# B&R Automation Studio project RS15_RX_30005_r00 (part 4)

#### A2_CycleCyclic.st
```iecst
(********************************************************************
 * COPYRIGHT -- .
 ********************************************************************
 * Program: A2_Cycle
 * File: A2_CycleCyclic.st
 * Author: Dominique
 * Created: October 15, 2011
 ********************************************************************
 * Implementation of program A2_Cycle
 ********************************************************************)

PROGRAM _CYCLIC

// Manu axis movement for timing setting

    //----------------------------------------------------------------------
    // FP Nip rolle auto Off
    // During timing setting automatique switch Off nip rolle
       stTON_02 (IN:=gstCycA[2].CycManTimSet.bCyc ,PT:=T#650ms) ;
       stTOF_00 (IN:=gstCycA[2].CycManTimSet.bCyc ,PT:=T#1s_500ms) ;
       g_bFP_NipRolAutoOff := gstCycA[2].CycManTimSet.bCyc OR
                              stTOF_00.Q                   ;

    //----------------------------------------------------------------------
    // Offset management

    // When synchro is off, Offset is set to 0
       IF NOT(gA[2].Ind_SynchronizedMotion) AND
          gstCycA[2].CycManTimSet.bFCyc     THEN
         rPrintRolActOffsetInch := 0.0 ;
         rSP_PrintRolOffsetInch := 0.0 ;
       END_IF ;
    // Set point Offset value Lock
    g_bLockSP_OffsetPrintRol := NOT(g_bCondManuTimSet)            OR
                                gstCycA[2].CycManTimSet.bSCyc     OR
                                0                                 ;

    // Offset Manu button animation
    bLockOffsetPB_Man := g_bFP_SP_Offset                   OR
                         g_bStartOffsetAuto                OR
                         NOT(g_bCondManuTimSet)            ;

    // Limit offset set point
    rSP_PrintRolOffsetInch := LIMIT(0.0,rSP_PrintRolOffsetInch,gRecipeActive.Repeat) ;
    IF gA[2].Cmd_ManuTimSetPlus THEN
      rSP_PrintRolOffsetInch := 0.0 ;
    END_IF ;
    // Calculation distance on axis
    rSP_AxisOffsetInch := rSP_PrintRolOffsetInch * gA[2].rRSynNum / gA[2].rRSynDen ;

    // Offset Auto button animation
    bLockOffsetPB := gstCycA[2].CycManTimSet.bFCyc     AND
                     (rSP_PrintRolOffsetInch <= 0.0)   OR
                     g_HMI_Cmd_ManuTimSetPlus          OR
                     (gstCycA[2].CycManTimSet.iStep>2) AND
                     NOT(g_bFP_SP_Offset)            ;

    IF NOT(bLockOffsetPB)        AND
       NOT(HMI_Cmd_AutoOffsetPB) THEN
      iAnimOffsetPB := 2 ;                     // Ready
    END_IF ;
    IF (rSP_PrintRolOffsetInch>0.0) AND
       NOT(g_bFP_SP_Offset)         AND
       NOT(bLockOffsetPB)           AND
       HMI_Cmd_AutoOffsetPB         THEN
      iAnimOffsetPB := 3 ;                     // Start
    END_IF ;
    IF g_bFP_SP_Offset THEN
      iAnimOffsetPB := 4 ;                     // Stop
    END_IF ;
    IF bLockOffsetPB THEN
      iAnimOffsetPB := 0 ;                     // PB Lock
    END_IF ;

    CASE iAnimOffsetPB OF
      0..1 : ; // PB Lock
        uiSP_OffsetCol_Ind := gBlue + gWhite * 256 ;
      2 : ;    // Ready
        uiSP_OffsetCol_Ind := gBlue + gWhite * 256 ;
      3 : ;    // Start
        uiSP_OffsetCol_Ind := gGreen + gBlack * 256 ;
      4 : ;    // Stop
        uiSP_OffsetCol_Ind := gRed + gBlack * 256 ;
    END_CASE
    uiSP_OffsetTxt_Ind := iAnimOffsetPB ;

    // Start Offset Auto
    IF EDGENEG(HMI_Cmd_AutoOffsetPB) THEN
      g_bStartOffsetAuto := 1 ;
    END_IF ;

    //---------------------------------------------------------------------------------------------------------------------
    // Printing rolle offset cycle
    //---------------------------------------------------------------------------------------------------------------------
    // Start cycle
    gstCycA[2].CycManTimSet.CmdStart := ( gA[2].Cmd_ManuTimSetPlus    OR
                                          gA[2].Cmd_ManuTimSetMinus ) AND
                                        gA[2].Ind_Ready               OR
                                        g_bStartOffsetAuto            AND
                                        1                             ;
    IF gstCycA[2].CycManTimSet.CmdStart THEN
      gstCycA[2].CycManTimSet.bSCyc := 1 ;
    END_IF ;

    //----------------------------------------------------------------------
    // Cycle at rest
    IF NOT(gstCycA[2].CycManTimSet.bSCyc) AND
       1                                  THEN
      IF NOT( gstCycA[2].CycManTimSet.bFCyc ) THEN
        // Init after cycle unpropaly ended
        gstCycA[2].CycManTimSet.bFCyc := 1 ;
        gstCycA[2].CycManTimSet.bCyc  := 0 ;

        g_bFP_SP_Offset                      := 0 ;
        g_bStartOffsetAuto                   := 0 ;
        gstCycA[2].CycManTimSet.CmdMov       := 0 ;
        gstCycA[2].CycManTimSet.CmdStop      := 0 ;
        gstCycA[2].CycManTimSet.CmdSynchroOn := 0 ;
        gstCycA[2].CycManTimSet.CmdExeMov    := 0 ;
        gstCycA[2].CycManTimSet.CmdExeStop   := 0 ;
      END_IF
      gstCycA[2].CycManTimSet.iStep := 0 ;
      RETURN ;
    ELSE
    //----------------------------------------------------------------------
    // Cycle running

      // Permanent conditions
      IF ( NOT(gA[2].Ind_Ready)                    OR
           NOT(gstCycA[2].CycManTimSet.CmdStart) ) AND
         NOT(g_bFP_SP_Offset)                      AND
         NOT(g_bStartOffsetAuto)                   AND
         (gstCycA[2].CycManTimSet.iStep <= 2)      THEN
        gstCycA[2].CycManTimSet.bSCyc := 0 ;
        RETURN ;
      END_IF

      IF g_bFP_SP_Offset                   AND
         ( NOT(gStopStringOK)              OR
           EDGEPOS(HMI_Cmd_AutoOffsetPB) ) THEN
        gstCycA[2].CycManTimSet.iStep := C_iSTEP_13 ;
        // Action Step 13
        gstCycA[2].CycManTimSet.CmdExeMov  := 0 ;
        gstCycA[2].CycManTimSet.CmdExeStop := 1 ;
        // Waiting Stop
      END_IF

      IF (gstCycA[2].CycManTimSet.iStep = C_iSTEP_11) AND
         (gstCycA[2].CycManTimSet.enMoveStat = FAULT) THEN
        gstCycA[2].CycManTimSet.iStep := C_iSTEP_16 ;
        // Action Step 16
        // Waiting Reset Fault
      END_IF

      // Permanent actions
      stTON_01 (
            IN := ( gstCycA[2].CycManTimSet.iStep = C_iSTEP_0 ) ,
            PT := T#30ms
               ) ;

      // Actual offset calculation
      IF (gstCycA[2].CycManTimSet.iStep >= C_iSTEP_3) THEN
        rTempDiffPrintRolPos := g_rPrintRolCalcPos_in - rMemoPosPrintRol ;
        rMemoPosPrintRol := g_rPrintRolCalcPos_in ;
        rDiffPrintRolPos := H_FC_Modulus (
                                 IN_rMod := gRecipeActive.Repeat ,
                                 IN_rVar := rTempDiffPrintRolPos
                                         ) ;
        rTempActOffsetInch[2] := rPrintRolActOffsetInch ;
        rPrintRolActOffsetInch := rPrintRolActOffsetInch + rDiffPrintRolPos ;
        rPrintRolActOffsetInch := H_FC_Modulus (
                                       IN_rMod := gRecipeActive.Repeat ,
                                       IN_rVar := rPrintRolActOffsetInch
                                               ) ;

        // Set point distance Offset animation
        IF g_bFP_SP_Offset THEN
          rSP_PrintRolOffsetInch := rSP_PrintRolOffsetInch - rDiffPrintRolPos ;
          IF (rSP_PrintRolOffsetInch < 0.001) THEN
            rSP_PrintRolOffsetInch := 0.0 ;
          END_IF
        END_IF
      END_IF

      stTON_03 (
            IN := (gstCycA[2].CycManTimSet.iStep = C_iSTEP_15) AND NOT(HMI_Cmd_AutoOffsetPB) ,
            PT := T#500ms
               ) ;

    END_IF
    //----------------------------------------------------------------------
    // Cycle steps

        CASE gstCycA[2].CycManTimSet.iStep OF

        C_iSTEP_0 :
         //----------------------------------------------
         // Etape 1 : Initialisation
         //           Waiting auto switch Off nip rolle
         //----------------------------------------------
          IF stTON_01.Q THEN
            gstCycA[2].CycManTimSet.iStep := C_iSTEP_1 ;

            // Action Step 1
            gstCycA[2].CycManTimSet.bFCyc := 0 ;
            gstCycA[2].CycManTimSet.bCyc  := 1 ;

            gstCycA[2].CycManTimSet.rSP_Distance := 0 ;
          END_IF

        C_iSTEP_1 :
         //----------------------------------------------
         // Etape 2  : Synchro
         //----------------------------------------------
          // Condition Step2
          IF (stTON_02.Q OR stTOF_00.Q) THEN
            gstCycA[2].CycManTimSet.iStep := C_iSTEP_2 ;

            // Action Step 2
            gstCycA[2].CycManTimSet.CmdSynchroOn := 1 ;
          END_IF

        C_iSTEP_2 :
         //----------------------------------------------
         // Step 3 : Activation motion and Stop waiting
         // Etape 10 : Synchro and start Offset with set point
         //----------------------------------------------
          IF gstCycA[2].CycManTimSet.bSynchroOkSlavA[2] AND
             (rSP_PrintRolOffsetInch <= 0)              THEN
            gstCycA[2].CycManTimSet.iStep := C_iSTEP_3 ;

            // Action Step 3
            gstCycA[2].CycManTimSet.CmdMov  := 1 ;
            gstCycA[2].CycManTimSet.CmdStop := 0 ;
            // Stop waiting
            // Memo printing cylinder actual position
            rMemoPosPrintRol := g_rPrintRolCalcPos_in ;
            RETURN ;
          END_IF
          // Condition Step10
          IF stTON_02.Q                                 AND
             gstCycA[2].CycManTimSet.bSynchroOkSlavA[2] AND
             g_bStartOffsetAuto                         AND
             ( gstCycA[2].CycManTimSet.bTestOn          OR
               NOT(gstCycA[2].CycManTimSet.bModTest) )  THEN
            gstCycA[2].CycManTimSet.iStep := C_iSTEP_10 ;

            // Action Step 10
            gstCycA[2].CycManTimSet.bTestOn := 0 ;

            g_bFP_SP_Offset    := 1 ;
            g_bStartOffsetAuto := 0 ;
            gstCycA[2].CycManTimSet.CmdExeMov  := 1 ;
            gstCycA[2].CycManTimSet.CmdExeStop := 0 ;
            gstCycA[2].CycManTimSet.rSP_Distance := rSP_AxisOffsetInch ;
            // Memo printing cylinder actual position
            rMemoPosPrintRol := g_rPrintRolCalcPos_in ;
          END_IF

        C_iSTEP_3 :
         //----------------------------------------------
         // Step 4 : Stop motion and End stop waiting
         //----------------------------------------------
          IF NOT(gstCycA[2].CycManTimSet.CmdStart) THEN
            gstCycA[2].CycManTimSet.iStep := C_iSTEP_4 ;

            // Action Step 4
            gstCycA[2].CycManTimSet.CmdMov  := 0 ;
            gstCycA[2].CycManTimSet.CmdStop := 1 ;
            // End stop waiting
          END_IF

        C_iSTEP_4 :
         //----------------------------------------------
         // Step 3 : Activation motion and Stop waiting
         // Step 5 : Cut synchro
         //----------------------------------------------
          // Condition Step3
          IF gstCycA[2].CycManTimSet.CmdStart THEN
            gstCycA[2].CycManTimSet.iStep := C_iSTEP_3 ;

            // Action Step 3
            gstCycA[2].CycManTimSet.CmdMov  := 1 ;
            gstCycA[2].CycManTimSet.CmdStop := 0 ;
            // Stop waiting
            RETURN ;
          END_IF ;
          // Condition Step5
          IF NOT(gstCycA[2].CycManTimSet.CmdStop) THEN
            gstCycA[2].CycManTimSet.iStep := C_iSTEP_5 ;

            // Action Step 5
            gstCycA[2].CycManTimSet.CmdSynchroOn := 0 ;
          END_IF

        C_iSTEP_5 :
         //----------------------------------------------
         // Step 0 : First step
         //----------------------------------------------
          IF TRUE THEN
            gstCycA[2].CycManTimSet.iStep := C_iSTEP_0 ;

            // Action Step 0
            gstCycA[2].CycManTimSet.bSCyc := 0 ;
            gstCycA[2].CycManTimSet.bFCyc := 1 ;
            gstCycA[2].CycManTimSet.bCyc  := 0 ;
          END_IF

        C_iSTEP_10 :
         //----------------------------------------------
         // Step 11 : Waiting end of move
         //----------------------------------------------
          IF TRUE                                          AND
             ( gstCycA[2].CycManTimSet.bTestOn             OR
               NOT(gstCycA[2].CycManTimSet.bModTest) )     THEN
            gstCycA[2].CycManTimSet.iStep := C_iSTEP_11 ;

            // Action Step 11
            gstCycA[2].CycManTimSet.bTestOn := 0 ;

            // Waiting end of move
          END_IF

        C_iSTEP_11 :
         //----------------------------------------------
         // Step 12 : End move
         //----------------------------------------------
          IF (gstCycA[2].CycManTimSet.enMoveStat = FINISHED) AND
             ( gstCycA[2].CycManTimSet.bTestOn               OR
               NOT(gstCycA[2].CycManTimSet.bModTest) )       THEN
            gstCycA[2].CycManTimSet.iStep := C_iSTEP_12 ;

            // Action Step 12
            gstCycA[2].CycManTimSet.bTestOn := 0 ;

            gstCycA[2].CycManTimSet.CmdExeMov := 0 ;
            g_bFP_SP_Offset := 0 ;
          END_IF

        C_iSTEP_12 :
         //----------------------------------------------
         // Step 0 : First step
         //----------------------------------------------
          IF (gstCycA[2].CycManTimSet.enMoveStat = INACTIVE) AND
             ( gstCycA[2].CycManTimSet.bTestOn               OR
               NOT(gstCycA[2].CycManTimSet.bModTest) )       THEN
            gstCycA[2].CycManTimSet.iStep := C_iSTEP_0 ;

            // Action Step 0
            gstCycA[2].CycManTimSet.bTestOn := 0 ;

            gstCycA[2].CycManTimSet.CmdSynchroOn := 0 ;

            gstCycA[2].CycManTimSet.bSCyc := 0 ;
            gstCycA[2].CycManTimSet.bFCyc := 1 ;
            gstCycA[2].CycManTimSet.bCyc  := 0 ;
          END_IF

        C_iSTEP_13 :
         //----------------------------------------------
         // Step 14 : End stop
         //----------------------------------------------
          IF (gstCycA[2].CycManTimSet.enMoveStat = INACTIVE) AND
             ( gstCycA[2].CycManTimSet.bTestOn               OR
               NOT(gstCycA[2].CycManTimSet.bModTest) )       AND
             gA[2].Ind_StandStill                            THEN
            gstCycA[2].CycManTimSet.iStep := C_iSTEP_14 ;

            // Action Step 14
            gstCycA[2].CycManTimSet.bTestOn := 0 ;

            gstCycA[2].CycManTimSet.CmdExeStop := 0 ;
          END_IF

        C_iSTEP_14 :
         //----------------------------------------------
         // Step 15 : Waiting
         //----------------------------------------------
          IF gA[2].Ind_SynchronizedMotion                  AND
             ( gstCycA[2].CycManTimSet.bTestOn             OR
               NOT(gstCycA[2].CycManTimSet.bModTest) )     THEN
            gstCycA[2].CycManTimSet.iStep := C_iSTEP_15 ;

            // Action Step 15
            gstCycA[2].CycManTimSet.bTestOn := 0 ;

            // Waiting
          END_IF

        C_iSTEP_15 :
         //----------------------------------------------
         // Step 0 : First step
         //----------------------------------------------
          IF stTON_03.Q                                    AND
             ( gstCycA[2].CycManTimSet.bTestOn             OR
               NOT(gstCycA[2].CycManTimSet.bModTest) )     THEN
            gstCycA[2].CycManTimSet.iStep := C_iSTEP_0 ;

            // Action Step 0
            gstCycA[2].CycManTimSet.bTestOn := 0 ;

            gstCycA[2].CycManTimSet.bSCyc := 0 ;
            gstCycA[2].CycManTimSet.bFCyc := 1 ;
            gstCycA[2].CycManTimSet.bCyc  := 0 ;
            g_bStartOffsetAuto := 0 ;
            g_bFP_SP_Offset    := 0 ;
            gstCycA[2].CycManTimSet.CmdSynchroOn := 0 ;
          END_IF

        C_iSTEP_16 :
         //----------------------------------------------
         // Step 17 : End cycle
         //----------------------------------------------
          IF gAlarmReset                                   AND
             ( gstCycA[2].CycManTimSet.bTestOn             OR
               NOT(gstCycA[2].CycManTimSet.bModTest) )     THEN
            gstCycA[2].CycManTimSet.iStep := C_iSTEP_17 ;

            // Action Step 17
            gstCycA[2].CycManTimSet.bTestOn := 0 ;

            gstCycA[2].CycManTimSet.CmdExeMov := 0 ;
          END_IF

        C_iSTEP_17 :
         //----------------------------------------------
         // Step 0 : First step
         //----------------------------------------------
          IF (gstCycA[2].CycManTimSet.enMoveStat = INACTIVE) AND
             ( gstCycA[2].CycManTimSet.bTestOn               OR
               NOT(gstCycA[2].CycManTimSet.bModTest) )       THEN
            gstCycA[2].CycManTimSet.iStep := C_iSTEP_0 ;

            // Action Step 0
            gstCycA[2].CycManTimSet.bTestOn := 0 ;

            gstCycA[2].CycManTimSet.bSCyc := 0 ;
            gstCycA[2].CycManTimSet.bFCyc := 1 ;
            gstCycA[2].CycManTimSet.bCyc  := 0 ;
            g_bStartOffsetAuto := 0 ;
            g_bFP_SP_Offset    := 0 ;
            gstCycA[2].CycManTimSet.CmdSynchroOn := 0 ;
          END_IF
        END_CASE
    //---------------------------------------------------------------------------------------------------------------------

END_PROGRAM
```

### Package Logical/BagMachine_Section/Holding - Axis

### Data object Logical/BagMachine_Section/Holding/Axis3/A3_Init (Ax) - Servo Axis Initialization File

#### A3_Init.ax
```
InitParameter (Version=2.24.0, NcSwId=ACP10)
  ACP10AXIS_typ:
    dig_in:
      level:
        reference = ncACTIV_HI
        pos_hw_end = ncACTIV_HI
        neg_hw_end = ncACTIV_HI
        trigger1 = ncACTIV_HI
        trigger2 = ncACTIV_HI
    encoder_if:
      parameter:
        count_dir = ncINVERSE
        scaling:
          load:
            units = 24000  // Units at the load = 36000 x 2 / 3
            rev_motor = 1  // Motor revolutions = 1
    limit:
      parameter:
        v_pos = 1.2e+006
        v_neg = 1.2e+006
        a1_pos = 5e+006
        a2_pos = 5e+006
        a1_neg = 5e+006
        a2_neg = 5e+006
        t_jolt = 0.0
        t_in_pos = 0.0
        pos_sw_end = 8388607
        neg_sw_end = -8388608
        ds_warning = 500.0
        ds_stop = 1000.0
        a_stop = 1e+030
        dv_stop = 0
        dv_stop_mode = ncOFF
    controller:
      mode = ncPOSITION
      position:
        kv = 300.0
        tn = 0.0
        t_predict = 0.0004
        t_total = 0.0012
        p_max = 1e+030
        i_max = 0.0
      speed:
        kv = 30.0
        tn = 0.0
        t_filter = 0.0
        isq_filter1:
          type = ncOFF
          a0 = 0.0
          a1 = 0.0
          b0 = 0.0
          b1 = 0.0
          b2 = 0.0
          c0_par_id = 0
          c1_par_id = 0
        isq_filter2:
          type = ncOFF
          a0 = 0.0
          a1 = 0.0
          b0 = 0.0
          b1 = 0.0
          b2 = 0.0
          c0_par_id = 0
          c1_par_id = 0
        isq_filter3:
          type = ncOFF
          a0 = 0.0
          a1 = 0.0
          b0 = 0.0
          b1 = 0.0
          b2 = 0.0
          c0_par_id = 0
          c1_par_id = 0
      uf:
        type = ncLINEAR
        auto_config = ncMOTOR_PAR
        u0 = 0.0
        un = 0.0
        fn = 50.0
        k_f_slip = 0.0
      ff:
        torque_load = 0.0
        torque_pos = 0.0
        torque_neg = 0.0
        kv_torque = 0.0
        inertia = 0.0
        t_filter_a = 0.0
    move:
      stop:
        parameter[0]:
          decel_ramp = ncA_LIMIT
          controller = ncON
        parameter[1]:
          decel_ramp = ncA_LIMIT
          controller = ncON
        parameter[2]:
          decel_ramp = ncA_LIMIT
          controller = ncON
        parameter[3]:
          decel_ramp = ncA_LIMIT
          controller = ncON
        quickstop:
          decel_ramp = ncA_LIMIT
        drive_error:
          decel_ramp = ncA_LIMIT
      homing:
        parameter:
          s = 0
          v_switch = 3600.0
          v_trigger = 360.0
          a = 50000.0
          mode = ncHOME_OFFSET
          edge_sw = ncNEGATIVE
          start_dir = ncNEGATIVE
          trigg_dir = ncNEGATIVE
          ref_pulse = ncOFF
          tr_s_block = 0.0
      basis:
        parameter:
          v_pos = 36000.0
          v_neg = 100000.0
          a1_pos = 50000.0
          a2_pos = 50000.0
          a1_neg = 50000.0
          a2_neg = 50000.0
    message:
      text:
        parameter:
          format = ncBREAK
          columns = 80
          data_modul = Error_Eng
```

### Data object Logical/BagMachine_Section/Holding/Axis3/A3_Par (Apt) - Servo Axis Parameter File

#### A3_Par.apt
```
AcoposParameterTable:
  Root Parameters:
    110 = ncSW_OFF (Name=CMD_SIMULATION)  // Simulation mode: Command
    128 = 1 (Name=SGEN_SW_END_IGNORE)  // SGEN_SW_END_IGNORE
    390 = 565 (Name=UDC_NOMINAL, Unit=V)  // CTRL DC bus: Nominal voltage
    944 = 464 (Name=REFERENCE_SWITCH_PARID)  // REFERENCE_SWITCH_PARID
```

### Program Logical/BagMachine_Section/Holding/Axis3/A3_Basic (IEC) - Basic Servo

#### A3_Basic.var - Local variables
```iecst
(********************************************************************
 * COPYRIGHT -- Microsoft
 ********************************************************************
 * Program: A3_Basic
 * File: A3_Basic.var
 * Author: pkiel
 * Created: July 13, 2011
 ********************************************************************
 * Local variables of program A3_Basic
 ********************************************************************)
VAR
	AutoAck : BOOL;
	AxisErrorNcAccess : UINT;
	DriveStatus : MC_DRIVESTATUS_TYP;
	HomeRestore : BOOL;
	InitEndlessPosition : BOOL;
	InitModPos_Done : BOOL;
	InitModPosition : BOOL;
	MC_BR_InitEndlessPosition_0 : MC_BR_InitEndlessPosition;
	MC_BR_InitModPos_0 : MC_BR_InitModPos;
  MC_BR_Phasing_0 : MC_BR_Phasing;
  MC_BR_Phasing_1 : MC_BR_Phasing;
	MC_BR_ReadDriveStatus_0 : MC_BR_ReadDriveStatus;
	MC_Home_0 : MC_Home;
	MC_Home_1 : MC_Home;
	MC_MoveVelocity_0 : MC_MoveVelocity;
	MC_Power_0 : MC_Power;
	MC_ReadActualPosition_0 : MC_ReadActualPosition;
	MC_ReadActualTorque_0 : MC_ReadActualTorque;
	MC_ReadActualVelocity_0 : MC_ReadActualVelocity;
	MC_ReadAxisError_0 : MC_ReadAxisError;
	MC_ReadStatus_0 : MC_ReadStatus;
	MC_Reset_0 : MC_Reset;
  MC_Stop_0 : MC_Stop;
  MC_Stop_1 : MC_Stop;

  MC_SetOverride_0 : MC_SetOverride ;
	ResetError : BOOL;
  rAxisTimSet_SP_Vel  : REAL ; (*Set point Velocity for Axis manual timing setting cycle, in units/s*)
  rAxisTimSet_SP_Acc  : REAL ; (*Set point Acceleration for Axis manual timing setting cycle, in units/s²*)
  rAxisTimSet_SP_Dec  : REAL ; (*Set point Deceleration for Axis manual timing setting cycle, in units/s²*)
  uiAxisTimSet_SP_Dir : USINT ; (*Set point Direction for Axis manual timing setting cycle*)
  uiAxisTimSet_SP_ShiftAppMode : UINT ; (*Set point Shit Application mode for phasing Axis manual timing setting cycle*)
  bTest_ : ARRAY[0..9] OF  BOOL;
  iTest_ : ARRAY[0..9] OF  INT;
  rTemp_ : ARRAY[0..9] OF REAL ;
  rTempActPhasDeg : REAL ;
  rTempActPhasDeg1 : REAL ;
  rTempActPhasDeg2 : REAL ;
  rTempAxisTimSet_SP_Acc : REAL;
  rTempAxisTimSet_SP_Dec : REAL;
  rPhasing_1_SP_Acc : REAL;
  rA9PosCorDeg  : REAL;
  rRepeatMetric : REAL;

  iiSP_SlPos_U  : DINT ; (*On Slave side, input set point position of the position controller ParID 428, in unit*)
  rSP_SlPos_Deg : REAL ; (*On Slave side, input set point position of the position controller ParID 428, in deg*)
  iiSP_MaPos_U  : DINT ; (*On Master side, input set point position of the position controller ParID 412, in unit*)
  rSP_MaPos_Deg : REAL ; (*On Master side, input set point position of the position controller ParID 412, in deg*)
  MC_BR_CyclicRead_0 : MC_BR_CyclicRead ;
  MC_BR_CyclicRead_1 : MC_BR_CyclicRead ;

  H_FB_RelativeChangeLimitReal_0 : H_FB_RelativeChangeLimitReal;
  rMin : REAL;
  IN_rRepeat : REAL;
  IN_rMin : REAL;
  IN_rMax : REAL;
  IN_bEnable : BOOL;
  rDiff : REAL;
  INOUT_rLimitIn : REAL;
  rOldLimitIn : REAL;
  rMax : REAL;
  rInput : REAL;
  IN_rInput : REAL;
  rOld : REAL;
  OUT_bChange : BOOL;
  OUT_rDiff : REAL;
  OUT_bOK : BOOL ;
  iIndex : INT ;
  rTempPosHolding : REAL ;
  st_TON_0 : TON;
  rSP_ShiftHolding   : REAL ;
  rSP_PhaseOffset    : REAL ;
  rSP_PhaseOffsetVal : REAL ;

  rA3PosTempAxis_deg : REAL ;
END_VAR
```

### Program Logical/BagMachine_Section/Holding/Axis3/A3_Control (IEC) - Servo Control

#### A3_Control.var
```iecst
(********************************************************************
 * COPYRIGHT -- Microsoft
 ********************************************************************
 * Program: A3_Control
 * File: A3_Control.var
 * Author: pkiel
 * Created: July 13, 2011
 ********************************************************************
 * Local variables of program A3_Control
 ********************************************************************)
VAR
	HGW_ChangeReal_0 : HGW_ChangeReal;
	HGW_RelativeChangeReal_0 : HGW_RelativeChangeReal;
  H_FB_RelativeChangeLimitReal1_0 : H_FB_RelativeChangeLimitReal1;
	HGW_Toggle_0 : HGW_Toggle;
	Synch_Permissive : BOOL;
	TOF_0 : TOF;
	TON_0 : TON;
  rIncrOffsetAxeRun_Inch : REAL ;
END_VAR
```

#### A3_ControlCyclic.ld
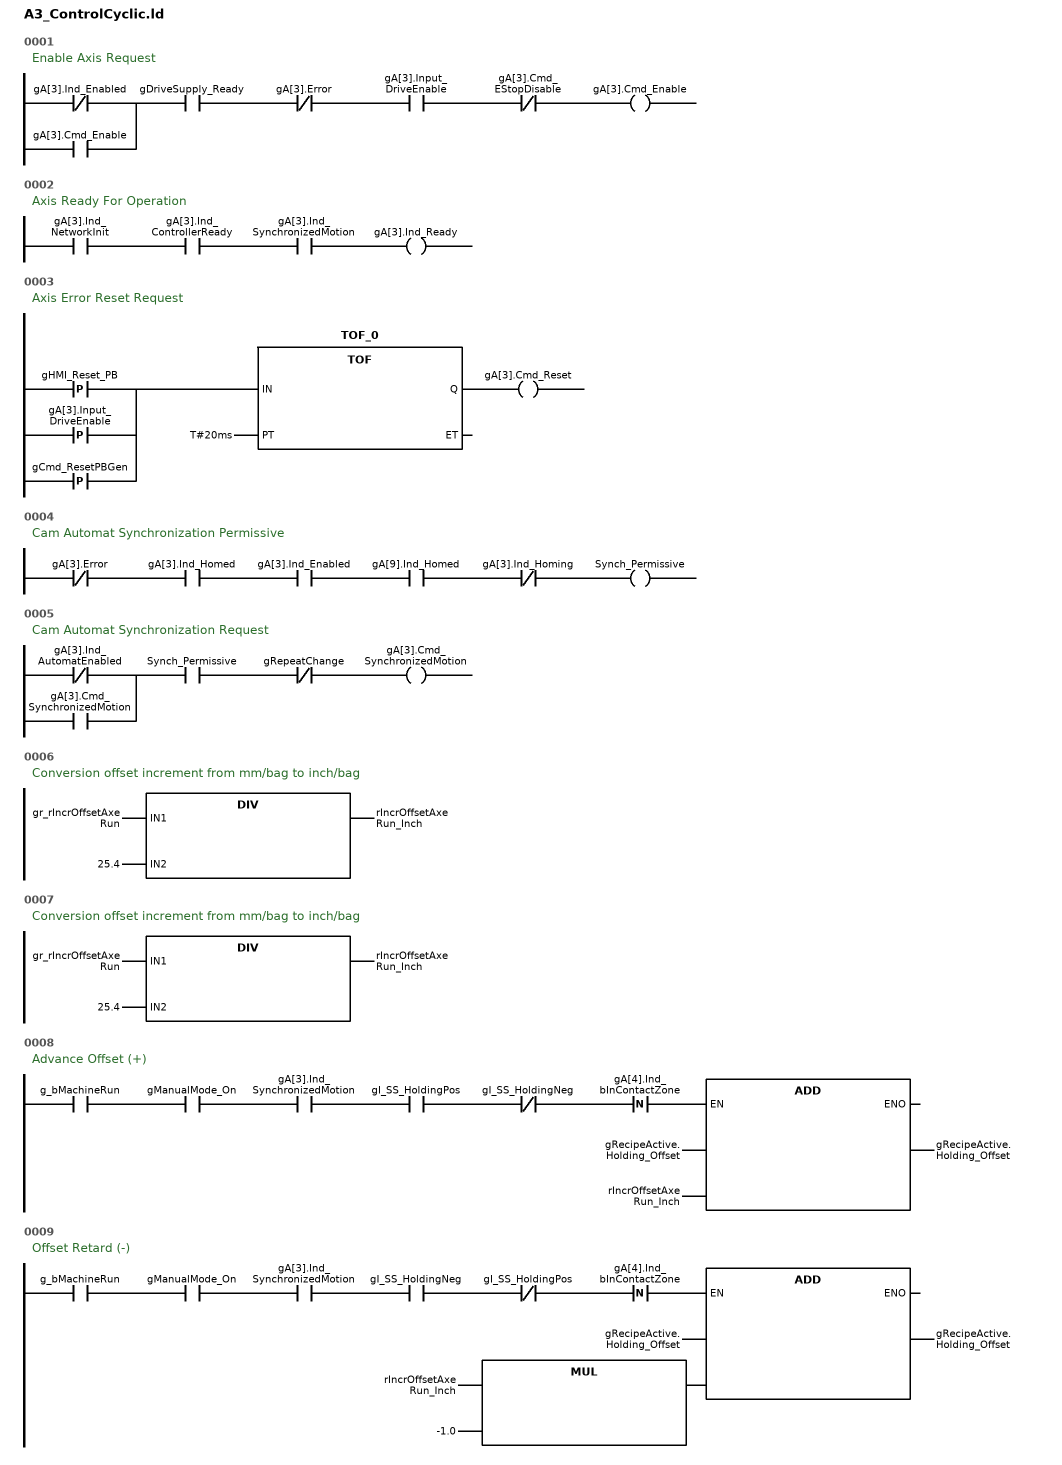
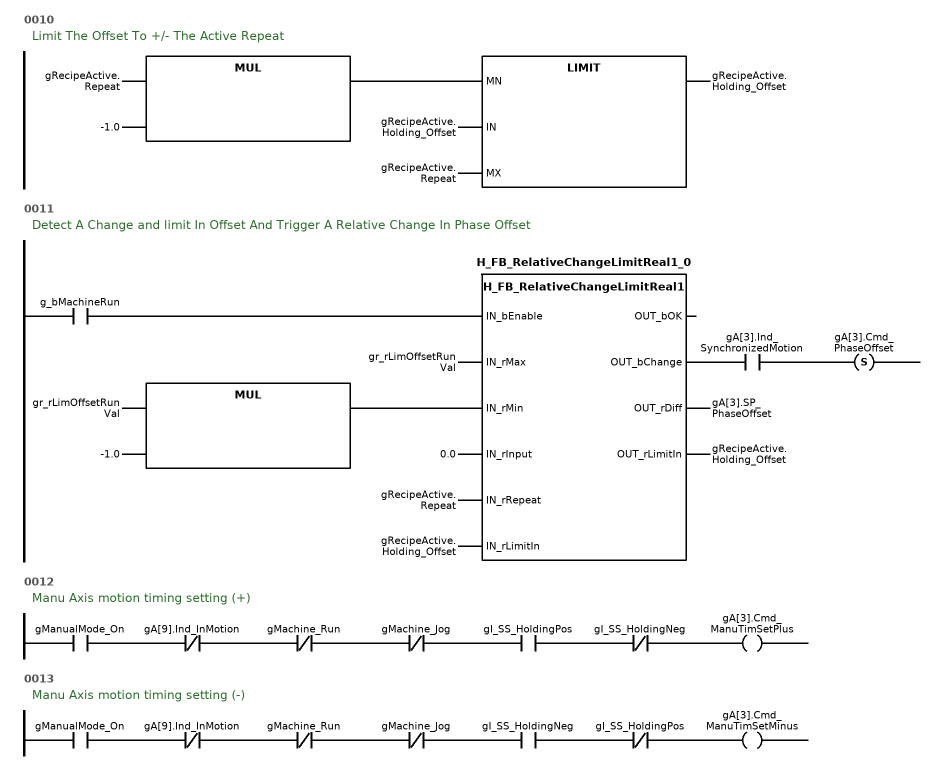
Ladder, written as Structured Text:
```iecst
(********************************************************************
 * COPYRIGHT -- Microsoft
 ********************************************************************
 * Program: A3_Control
 * File: A3_ControlCyclic.ld
 * Author: pkiel
 * Created: July 13, 2011
 ********************************************************************
 * Implementation of program A3_Control
 ********************************************************************)

PROGRAM _CYCLIC
VAR
    _e1 : R_TRIG;
    _e2 : R_TRIG;
    _e3 : R_TRIG;
    _e4 : F_TRIG;
    _e5 : F_TRIG;
END_VAR
(* Network 1: Enable Axis Request *)
gA[3].Cmd_Enable := (NOT gA[3].Ind_Enabled OR gA[3].Cmd_Enable) AND gDriveSupply_Ready AND NOT gA[3].Error AND gA[3].Input_DriveEnable AND NOT gA[3].Cmd_EStopDisable;

(* Network 2: Axis Ready For Operation *)
gA[3].Ind_Ready := gA[3].Ind_NetworkInit AND gA[3].Ind_ControllerReady AND gA[3].Ind_SynchronizedMotion;

(* Network 3: Axis Error Reset Request *)
_e1(CLK := gHMI_Reset_PB);
_e2(CLK := gA[3].Input_DriveEnable);
_e3(CLK := gCmd_ResetPBGen);
TOF_0(IN := _e1.Q OR _e2.Q OR _e3.Q, PT := T#20ms);
gA[3].Cmd_Reset := TOF_0.Q;

(* Network 4: Cam Automat Synchronization Permissive *)
Synch_Permissive := NOT gA[3].Error AND gA[3].Ind_Homed AND gA[3].Ind_Enabled AND gA[9].Ind_Homed AND NOT gA[3].Ind_Homing;

(* Network 5: Cam Automat Synchronization Request *)
gA[3].Cmd_SynchronizedMotion := (NOT gA[3].Ind_AutomatEnabled OR gA[3].Cmd_SynchronizedMotion) AND Synch_Permissive AND NOT gRepeatChange;

(* Network 6: Conversion offset increment from mm/bag to inch/bag *)
rIncrOffsetAxeRun_Inch := gr_rIncrOffsetAxeRun / 25.4;

(* Network 7: Conversion offset increment from mm/bag to inch/bag *)
rIncrOffsetAxeRun_Inch := gr_rIncrOffsetAxeRun / 25.4;

(* Network 8: Advance Offset (+) *)
_e4(CLK := gA[4].Ind_bInContactZone);
IF g_bMachineRun AND gManualMode_On AND gA[3].Ind_SynchronizedMotion AND gI_SS_HoldingPos AND NOT gI_SS_HoldingNeg AND _e4.Q THEN
    gRecipeActive.Holding_Offset := gRecipeActive.Holding_Offset + rIncrOffsetAxeRun_Inch;
END_IF;

(* Network 9: Offset Retard (-) *)
_e5(CLK := gA[4].Ind_bInContactZone);
IF g_bMachineRun AND gManualMode_On AND gA[3].Ind_SynchronizedMotion AND gI_SS_HoldingNeg AND NOT gI_SS_HoldingPos AND _e5.Q THEN
    gRecipeActive.Holding_Offset := gRecipeActive.Holding_Offset + (rIncrOffsetAxeRun_Inch * -1.0);
END_IF;

(* Network 10: Limit The Offset To +/- The Active Repeat *)
gRecipeActive.Holding_Offset := LIMIT(MN := gRecipeActive.Repeat * -1.0, IN := gRecipeActive.Holding_Offset, MX := gRecipeActive.Repeat);

(* Network 11: Detect A Change and limit In Offset And Trigger A Relative Change In Phase Offset *)
H_FB_RelativeChangeLimitReal1_0(IN_bEnable := g_bMachineRun, IN_rMax := gr_rLimOffsetRunVal, IN_rMin := gr_rLimOffsetRunVal * -1.0, IN_rInput := 0.0, IN_rRepeat := gRecipeActive.Repeat, IN_rLimitIn := gRecipeActive.Holding_Offset);
IF H_FB_RelativeChangeLimitReal1_0.OUT_bChange AND gA[3].Ind_SynchronizedMotion THEN
    gA[3].Cmd_PhaseOffset := TRUE;
END_IF;
gA[3].SP_PhaseOffset := H_FB_RelativeChangeLimitReal1_0.OUT_rDiff;
gRecipeActive.Holding_Offset := H_FB_RelativeChangeLimitReal1_0.OUT_rLimitIn;

(* Network 12: Manu Axis motion timing setting (+) *)
gA[3].Cmd_ManuTimSetPlus := gManualMode_On AND NOT gA[9].Ind_InMotion AND NOT gMachine_Run AND NOT gMachine_Jog AND gI_SS_HoldingPos AND NOT gI_SS_HoldingNeg;

(* Network 13: Manu Axis motion timing setting (-) *)
gA[3].Cmd_ManuTimSetMinus := gManualMode_On AND NOT gA[9].Ind_InMotion AND NOT gMachine_Run AND NOT gMachine_Jog AND gI_SS_HoldingNeg AND NOT gI_SS_HoldingPos;
END_PROGRAM
```

- Program Logical/BagMachine_Section/Holding/Axis3/A3_Automat (IEC) - Cam Automat (no source held here)

### Program Logical/BagMachine_Section/Holding/Axis3/A3_Ref (IEC) - Reference Routine

#### A3_Ref.var - Local variables
```iecst
(********************************************************************
 * COPYRIGHT -- Microsoft
 ********************************************************************
 * Program: A3_Ref
 * File: A3_Ref.var
 * Author: pkiel
 * Created: July 19, 2011
 ********************************************************************
 * Local variables of program A3_Ref
 ********************************************************************)
VAR
	HGW_2StepMove_0 : HGW_2StepMove;
	MC_Home_0 : MC_Home;
	MC_Home_1 : MC_Home;
	MC_MoveAdditive_0 : MC_MoveAdditive;
	Ref_Seq : ARRAY[0..10] OF BOOL;
  rDirection : REAL ;
END_VAR
```

### Program Logical/BagMachine_Section/Holding/Axis3/A3_Cycle (IEC) - A new program

#### A3_CycleCyclic.st - Cyclic code
```iecst
(********************************************************************
 * COPYRIGHT -- .
 ********************************************************************
 * Program: A1_Cycle
 * File: A1_CycleCyclic.st
 * Author: dominique
 * Created: August 01, 2011
 ********************************************************************
 * Implementation of program A1_Cycle
 ********************************************************************)

PROGRAM _CYCLIC

// Manu axis movement for timing setting

    //---------------------------------------------------------------------------------------------------------------------
    // Holding timing setting cycle
    //---------------------------------------------------------------------------------------------------------------------

    // Start cycle
    gstCycA[3].CycManTimSet.CmdStart := ( gA[3].Cmd_ManuTimSetPlus        OR
                                          gA[3].Cmd_ManuTimSetMinus )     AND
                                        ( NOT(g_bCycManTimeSetOn)         OR
                                          gstCycA[3].CycManTimSet.bSCyc ) AND
                                        gA[3].Ind_Ready                   AND
                                        gA[4].Ind_Ready                   AND
                                        gA[7].Ind_Ready                   ;
    IF gstCycA[3].CycManTimSet.CmdStart THEN
      gstCycA[3].CycManTimSet.bSCyc := 1 ;
    END_IF ;

    //----------------------------------------------------------------------
    // Cycle at rest
    IF NOT(gstCycA[3].CycManTimSet.bSCyc) AND
       1                                 THEN
      IF NOT( gstCycA[3].CycManTimSet.bFCyc ) THEN
        // Init after cycle unpropaly ended
        gstCycA[3].CycManTimSet.bFCyc := 1 ;
        gstCycA[3].CycManTimSet.bCyc  := 0 ;

        gstCycA[3].CycManTimSet.CmdMov       := 0 ;
        gstCycA[3].CycManTimSet.CmdStop      := 0 ;
        gstCycA[3].CycManTimSet.CmdSynchroOn := 0 ;

        gA[3].Cmd_Override  := 1 ;
        gA[3].rSP_OverrideA := 1.0 ;
      END_IF
      gstCycA[3].CycManTimSet.iStep := 0 ;
      RETURN ;
    ELSE
    //----------------------------------------------------------------------
    // Cycle running

      // Permanent conditions
      IF NOT(gA[3].Ind_Ready)                  OR
         NOT(gA[4].Ind_Ready)                  OR
         NOT(gA[7].Ind_Ready)                  OR
         NOT(gstCycA[3].CycManTimSet.CmdStart) AND
         (gstCycA[3].CycManTimSet.iStep <= 1)  THEN
        gstCycA[3].CycManTimSet.bSCyc := 0 ;
        RETURN ;
      END_IF

      // Permanent actions
      stTON_01 (
            IN := ( gstCycA[3].CycManTimSet.iStep = C_iSTEP_0 ) ,
            PT := T#30ms
               ) ;

      // Phasing override acce management ( Override seems do be not efficient with phasing )
      IF EDGE(gstCycA[3].CycManTimSet.CmdStart) THEN
        IF gstCycA[3].CycManTimSet.CmdStart THEN
          gA[3].rSP_OverrideA := 0.5 ;
        ELSE
          gA[3].rSP_OverrideA := 1.0 ;
        END_IF
        gA[3].Cmd_Override := 1 ;
      END_IF

    END_IF
    //----------------------------------------------------------------------
    // Cycle steps

        CASE gstCycA[3].CycManTimSet.iStep OF

        C_iSTEP_0 :
         //----------------------------------------------
         // Etape 1 : Initialisation
         //----------------------------------------------
          IF stTON_01.Q THEN
            gstCycA[3].CycManTimSet.iStep := C_iSTEP_1 ;

            // Action Step 1
            gstCycA[3].CycManTimSet.bFCyc := 0 ;
            gstCycA[3].CycManTimSet.bCyc  := 1 ;
          END_IF

        C_iSTEP_1 :
         //----------------------------------------------
         // Etape 2 : Synchro Tearing + Drum on Holding
         //----------------------------------------------
          IF TRUE THEN
            gstCycA[3].CycManTimSet.iStep := C_iSTEP_2 ;

            // Action Step 2
            gstCycA[3].CycManTimSet.CmdSynchroOn := 1 ;
          END_IF

        C_iSTEP_2 :
         //----------------------------------------------
         // Step 3 : Activation motion and Stop waiting
         // Step 6 : Exit cycle
         //----------------------------------------------
          // Condition Step3
          IF gstCycA[3].CycManTimSet.bSynchroOkSlavA[3]    AND
             gstCycA[3].CycManTimSet.bSynchroOkSlavA[4]    AND
             gstCycA[3].CycManTimSet.bSynchroOkSlavA[7]    AND
             ( gstCycA[3].CycManTimSet.bSynchroOkSlavA[12] OR
               NOT(gA[12].bInMach) )                       AND
             ( gstCycA[3].CycManTimSet.bSynchroOkSlavA[13] OR
               NOT(gA[13].bInMach) )                       AND
             NOT(gA[3].Cmd_Override)                       THEN
            gstCycA[3].CycManTimSet.iStep := C_iSTEP_3 ;

            // Action Step 3
            gstCycA[3].CycManTimSet.CmdMov  := 1 ;
            gstCycA[3].CycManTimSet.CmdStop := 0 ;
            // Stop waiting
            RETURN ;
          END_IF

          // Condition Step6
          IF NOT(gstCycA[3].CycManTimSet.CmdStart) THEN
            gstCycA[3].CycManTimSet.iStep := C_iSTEP_6 ;

            // Action Step 6
            gstCycA[3].CycManTimSet.CmdSynchroOn := 0 ;
          END_IF

        C_iSTEP_3 :
         //----------------------------------------------
         // Step 4 : Stop motion and End stop waiting
         //----------------------------------------------
          IF NOT(gstCycA[3].CycManTimSet.CmdStart) AND
             NOT(gA[3].Cmd_Override)               THEN
            gstCycA[3].CycManTimSet.iStep := C_iSTEP_4 ;

            // Action Step 4
            gstCycA[3].CycManTimSet.CmdMov  := 0 ;
            gstCycA[3].CycManTimSet.CmdStop := 1 ;
            // End stop waiting
          END_IF

        C_iSTEP_4 :
         //----------------------------------------------
         // Step 3 : Activation motion and Stop waiting
         // Step 5 : Cut synchro
         //----------------------------------------------
          // Condition Step3
          IF gstCycA[3].CycManTimSet.CmdStart AND
             NOT(gA[3].Cmd_Override)          THEN
            gstCycA[3].CycManTimSet.iStep := C_iSTEP_3 ;

            // Action Step 3
            gstCycA[3].CycManTimSet.CmdMov  := 1 ;
            gstCycA[3].CycManTimSet.CmdStop := 0 ;
            // Stop waiting
            RETURN ;
          END_IF
          // Condition Step5
          IF NOT(gstCycA[3].CycManTimSet.CmdStop) THEN
            gstCycA[3].CycManTimSet.iStep := C_iSTEP_5 ;

            // Action Step 5
            gstCycA[3].CycManTimSet.CmdSynchroOn := 0 ;
          END_IF

        C_iSTEP_5 :
         //----------------------------------------------
         // Step 6 : New offset calculation
         //----------------------------------------------
          IF NOT(gstCycA[3].CycManTimSet.bSynchroOkSlavA[4])    AND
             NOT(gstCycA[3].CycManTimSet.bSynchroOkSlavA[7])    AND
             ( NOT(gstCycA[3].CycManTimSet.bSynchroOkSlavA[12]) OR
               NOT(gA[12].bInMach) )                            AND
             ( NOT(gstCycA[3].CycManTimSet.bSynchroOkSlavA[13]) OR
               NOT(gA[13].bInMach) )                            THEN
            gstCycA[3].CycManTimSet.iStep := C_iSTEP_6 ;

            // Action Step 6
            // Memo Actual phase Offset
            rTempActPhasDeg[3] := gRecipeActive.rHolding_PhasMasterDeg ;
            rTempActOffsetInch[3] := gRecipeActive.Holding_Offset ;
            // Update phase
            gRecipeActive.rHolding_PhasMasterDeg := gA[3].rActPhasDeg ;
            gRecipeActive.rTearing_PhasMasterDeg := gA[4].rActPhasDeg ;
            gRecipeActive.rDrum_PhasMasterDeg    := gA[7].rActPhasDeg ;
            IF gA[12].bInMach THEN
              gRecipeActive.rEnvB_PhasMasterDeg := gA[12].rActPhasDeg ;
            END_IF
            IF gA[13].bInMach THEN
              gRecipeActive.rTearEB_PhasMasterDeg := gA[13].rActPhasDeg ;
            END_IF
            // Update Offset
            rTemp_[3] := rTempActOffsetInch[3] + (gRecipeActive.rHolding_PhasMasterDeg - rTempActPhasDeg[3])/(gA[3].rRSynNum/gA[3].rRSynDen)*gA[3].InchPerDeg ;
            gRecipeActive.Holding_Offset := H_FC_Modulus (IN_rMod := gRecipeActive.Repeat, IN_rVar := rTemp_[3]) ;
          END_IF

        C_iSTEP_6 :
         //----------------------------------------------
         // Step 0 : First step
         //----------------------------------------------
          IF NOT(gstCycA[3].CycManTimSet.bSynchroOkSlavA[4])    AND
             NOT(gstCycA[3].CycManTimSet.bSynchroOkSlavA[7])    AND
             ( NOT(gstCycA[3].CycManTimSet.bSynchroOkSlavA[12]) OR
               NOT(gA[12].bInMach) )                            AND
             ( NOT(gstCycA[3].CycManTimSet.bSynchroOkSlavA[13]) OR
               NOT(gA[13].bInMach) )                            THEN
            gstCycA[3].CycManTimSet.iStep := C_iSTEP_0 ;

            // Action Step 0
            gstCycA[3].CycManTimSet.bSCyc := 0 ;
            gstCycA[3].CycManTimSet.bFCyc := 1 ;
            gstCycA[3].CycManTimSet.bCyc  := 0 ;
          END_IF
        END_CASE
    //---------------------------------------------------------------------------------------------------------------------

END_PROGRAM
```

#### A3_CycleInit.st - Initialization code
```iecst
(********************************************************************
 * COPYRIGHT -- .
 ********************************************************************
 * Program: A3_Cycle
 * File: A3_CycleInit.st
 * Author: dominique
 * Created: August 01, 2011
 ********************************************************************
 * Implementation of program A1_Cycle
 ********************************************************************)

PROGRAM _INIT

  gstCycA[3].CycManTimSet.uiMasterParID := 428 ; // ParID 428 = CTRL Position controller: Input set position (in case real axis)

END_PROGRAM
```

### Package Logical/BagMachine_Section/Tearing - Axis

### Data object Logical/BagMachine_Section/Tearing/Axis4/A4_Init (Ax) - Servo Axis Initialization File

#### A4_Init.ax
```
InitParameter (Version=2.24.0, NcSwId=ACP10)
  ACP10AXIS_typ:
    dig_in:
      level:
        reference = ncACTIV_HI
        pos_hw_end = ncACTIV_HI
        neg_hw_end = ncACTIV_HI
        trigger1 = ncACTIV_HI
        trigger2 = ncACTIV_HI
    encoder_if:
      parameter:
        count_dir = ncSTANDARD
        scaling:
          load:
            units = 18000  // Units at the load     = 36000 / 2
            rev_motor = 1  // Motor revolutions    = 1
    limit:
      parameter:
        v_pos = 1.03e+006
        v_neg = 1.03e+006
        a1_pos = 5e+006
        a2_pos = 5e+006
        a1_neg = 5e+006
        a2_neg = 5e+006
        t_jolt = 0.0
        t_in_pos = 0.0
        pos_sw_end = 8388607
        neg_sw_end = -8388608
        ds_warning = 500.0
        ds_stop = 1000.0
        a_stop = 1e+030
        dv_stop = 0
        dv_stop_mode = ncOFF
    controller:
      mode = ncPOSITION
      position:
        kv = 300.0
        tn = 0.0
        t_predict = 0.0004
        t_total = 0.0012
        p_max = 1e+030
        i_max = 0.0
      speed:
        kv = 30.0
        tn = 0.0
        t_filter = 0.0
        isq_filter1:
          type = ncOFF
          a0 = 0.0
          a1 = 0.0
          b0 = 0.0
          b1 = 0.0
          b2 = 0.0
          c0_par_id = 0
          c1_par_id = 0
        isq_filter2:
          type = ncOFF
          a0 = 0.0
          a1 = 0.0
          b0 = 0.0
          b1 = 0.0
          b2 = 0.0
          c0_par_id = 0
          c1_par_id = 0
        isq_filter3:
          type = ncOFF
          a0 = 0.0
          a1 = 0.0
          b0 = 0.0
          b1 = 0.0
          b2 = 0.0
          c0_par_id = 0
          c1_par_id = 0
      uf:
        type = ncLINEAR
        auto_config = ncMOTOR_PAR
        u0 = 0.0
        un = 0.0
        fn = 50.0
        k_f_slip = 0.0
      ff:
        torque_load = 0.0
        torque_pos = 0.0
        torque_neg = 0.0
        kv_torque = 0.0
        inertia = 0.0
        t_filter_a = 0.0
    move:
      stop:
        parameter[0]:
          decel_ramp = ncA_LIMIT
          controller = ncON
        parameter[1]:
          decel_ramp = ncA_LIMIT
          controller = ncON
        parameter[2]:
          decel_ramp = ncA_LIMIT
          controller = ncON
        parameter[3]:
          decel_ramp = ncA_LIMIT
          controller = ncON
        quickstop:
          decel_ramp = ncA_LIMIT
        drive_error:
          decel_ramp = ncA_LIMIT
      homing:
        parameter:
          s = 0
          v_switch = 7200.0
          v_trigger = 720.0
          a = 50000.0
          mode = ncHOME_OFFSET
          edge_sw = ncPOSITIVE
          start_dir = ncPOSITIVE
          trigg_dir = ncPOSITIVE
          ref_pulse = ncOFF
          tr_s_block = 0.0
      basis:
        parameter:
          v_pos = 36000.0
          v_neg = 100000.0
          a1_pos = 50000.0
          a2_pos = 50000.0
          a1_neg = 50000.0
          a2_neg = 50000.0
    message:
      text:
        parameter:
          format = ncBREAK
          columns = 80
          data_modul = Error_Eng
```

### Data object Logical/BagMachine_Section/Tearing/Axis4/A4_Par (Apt) - Servo Axis Parameter File

#### A4_Par.apt
```
AcoposParameterTable:
  Root Parameters:
    110 = ncSW_OFF (Name=CMD_SIMULATION)  // Simulation mode: Command
    128 = 1 (Name=SGEN_SW_END_IGNORE)  // SGEN_SW_END_IGNORE
    390 = 565 (Name=UDC_NOMINAL, Unit=V)  // CTRL DC bus: Nominal voltage
    944 = 463 (Name=REFERENCE_SWITCH_PARID)  // REFERENCE_SWITCH_PARID
```

### Program Logical/BagMachine_Section/Tearing/Axis4/A4_Basic (IEC) - Basic Servo

#### A4_BasicInit.st - Initialization code
```iecst
(********************************************************************
 * COPYRIGHT -- Microsoft
 ********************************************************************
 * Program: A4_Basic
 * File: A4_BasicInit.st
 * Author: pkiel
 * Created: July 13, 2011
 ********************************************************************
 * Implementation of program A4_Basic
 ********************************************************************)

PROGRAM _INIT

	(* Axis Setpoint Variables *)
		gA[4].SP_MotorPPR := 18000 ;
		gA[4].SP_GearBoxInput:= 2;
    gA[4].SP_GearBoxOutput:= 1;
    gA[4].AxisPeriod := (gA[4].SP_MotorPPR*gA[4].SP_GearBoxInput/gA[4].SP_GearBoxOutput);
		gA[4].UnitsPerDeg := gA[4].AxisPeriod/360;
		gA[4].SP_Accel := 0.2*gA[4].AxisPeriod;
		gA[4].SP_Decel := 0.4*gA[4].AxisPeriod;
		gA[4].SP_EStopDecel := 1000.0*gA[4].AxisPeriod; // Stop axis from 1000 tr/min in 1s
		gA[4].HomeVelocity := 6*gA[4].AxisPeriod/60;
    gA[4].rSP_CorPosVel := 0.0 ;
    gA[4].rSP_OverrideV := 1.0 ;
    gA[4].rSP_OverrideA := 1.0 ;
    gA[4].Cmd_EStopDisable := 0 ;

	(* access master axis *)
		AxisErrorNcAccess := ncaccess(ncACP10MAN, ADR('Axis4'), ADR(gA[4].Ident));

	(* Trigger Initialization Of ModPosition *)
		InitModPosition:=1;

  // General parameter init
  gr_rTearAxContactZone := 52.0 ;

END_PROGRAM
```

#### A4_Basic.var - Local variables
```iecst
(********************************************************************
 * COPYRIGHT -- Microsoft
 ********************************************************************
 * Program: A4_Basic
 * File: A4_Basic.var
 * Author: pkiel
 * Created: July 13, 2011
 ********************************************************************
 * Local variables of program A4_Basic
 ********************************************************************)
VAR
	AutoAck : BOOL;
	AxisErrorNcAccess : UINT;
	DriveStatus : MC_DRIVESTATUS_TYP;
	HomeRestore : BOOL;
	InitEndlessPosition : BOOL;
	InitModPos_Done : BOOL;
	InitModPosition : BOOL;
	MC_BR_InitEndlessPosition_0 : MC_BR_InitEndlessPosition;
	MC_BR_InitModPos_0 : MC_BR_InitModPos;
  uiInitModPos0_ErrorID : UINT ;
  MC_BR_Phasing_0 : MC_BR_Phasing;
  MC_BR_Phasing_1 : MC_BR_Phasing;
	MC_BR_ReadDriveStatus_0 : MC_BR_ReadDriveStatus;
	MC_Home_0 : MC_Home;
  MC_Home_1 : MC_Home;
  MC_Home_2 : MC_Home;
	MC_MoveVelocity_0 : MC_MoveVelocity;
	MC_Power_0 : MC_Power;
	MC_ReadActualPosition_0 : MC_ReadActualPosition;
	MC_ReadActualTorque_0 : MC_ReadActualTorque;
	MC_ReadActualVelocity_0 : MC_ReadActualVelocity;
	MC_ReadAxisError_0 : MC_ReadAxisError;
	MC_ReadStatus_0 : MC_ReadStatus;
	MC_Reset_0 : MC_Reset;
  MC_Stop_0 : MC_Stop;
  MC_Stop_1 : MC_Stop;
  st_TON_0 : TON ;
	ResetError : BOOL;
  rAxisTimSet_SP_Vel  : REAL ; (*Set point Velocity for Axis manual timing setting cycle, in units/s*)
  rAxisTimSet_SP_Acc  : REAL ; (*Set point Acceleration for Axis manual timing setting cycle, in units/s²*)
  rAxisTimSet_SP_Dec  : REAL ; (*Set point Deceleration for Axis manual timing setting cycle, in units/s²*)
  uiAxisTimSet_SP_Dir : USINT ; (*Set point Direction for Axis manual timing setting cycle*)
  uiAxisTimSet_SP_ShiftAppMode : UINT ; (*Set point Shit Application mode for phasing Axis manual timing setting cycle*)
  rTempActPhasDeg : REAL;
  iTest_ : ARRAY[0..9] OF INT ;
  rTest_ : ARRAY[0..9] OF REAL ;
  rTemp_ : ARRAY[0..9] OF REAL ;
  iIndx : INT ;
  rA9PosCorDeg  : REAL;
  rRepeatMetric : REAL;
  MC_SetOverride_0 : MC_SetOverride;

  iiSP_SlPos_U  : DINT ; (*On Slave side, input set point position of the position controller ParID 428, in unit*)
  rSP_SlPos_Deg : REAL ; (*On Slave side, input set point position of the position controller ParID 428, in deg*)
  iiSP_MaPos_U  : DINT ; (*On Master side, input set point position of the position controller ParID 412, in unit*)
  rSP_MaPos_Deg : REAL ; (*On Master side, input set point position of the position controller ParID 412, in deg*)
  MC_BR_CyclicRead_0 : MC_BR_CyclicRead ;
  MC_BR_CyclicRead_1 : MC_BR_CyclicRead ;

  bChangeModReq      : BOOL ;
  rRedefPosTear      : REAL ;
  rPosTear4Pliers    : REAL ;
  rSP_PhaseOffset    : REAL ;
  rSP_PhaseOffsetVal : REAL ;
  rSP_ShiftTearing   : REAL ;
END_VAR
```

### Program Logical/BagMachine_Section/Tearing/Axis4/A4_Control (IEC) - Servo Control

#### A4_ControlCyclic.ld - Cyclic code
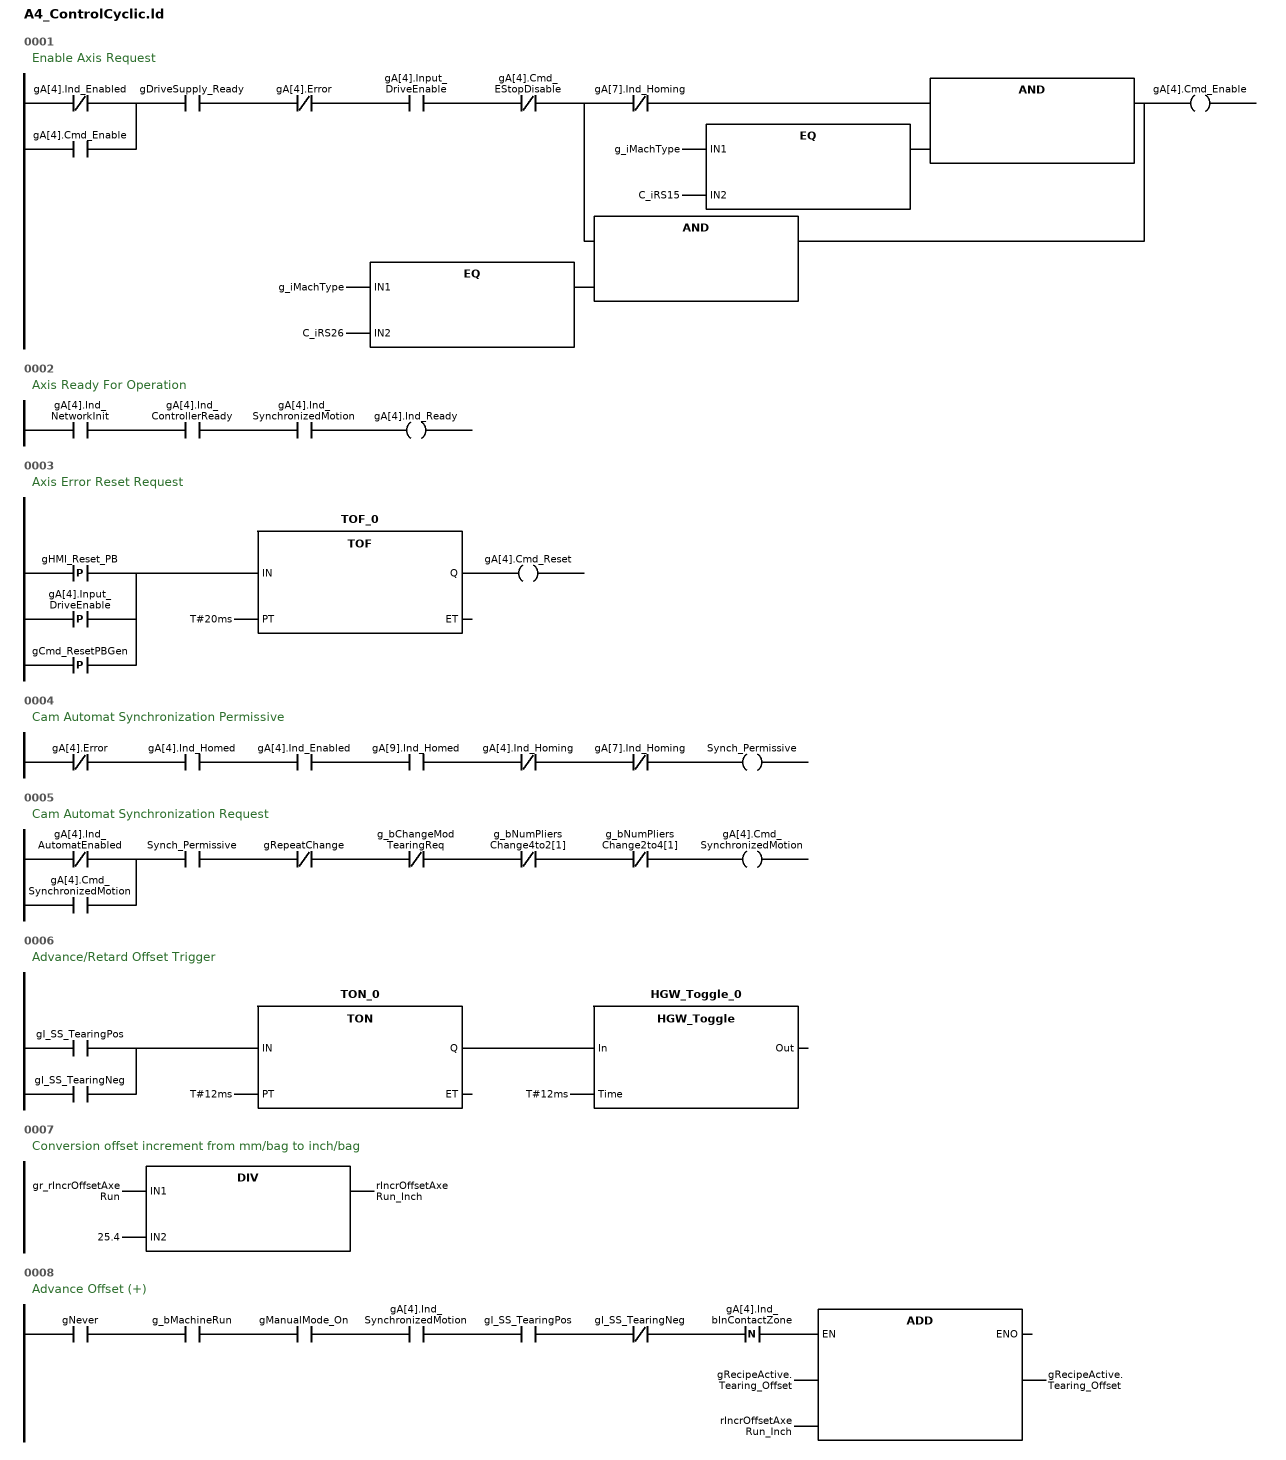
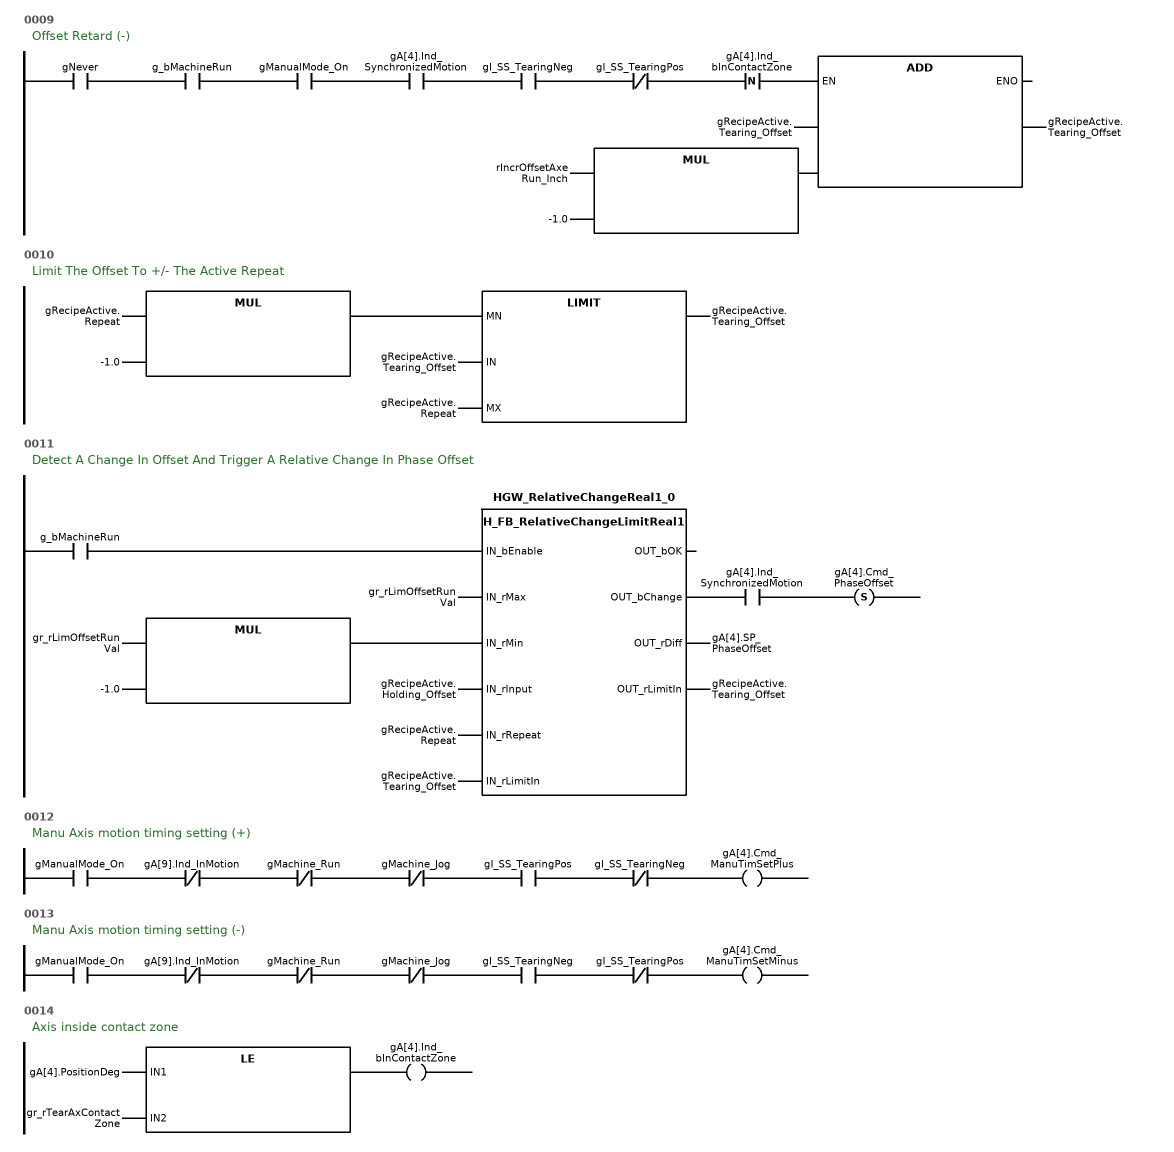
Ladder, written as Structured Text:
```iecst
(********************************************************************
 * COPYRIGHT -- Microsoft
 ********************************************************************
 * Program: A4_Control
 * File: A4_ControlCyclic.ld
 * Author: pkiel
 * Created: July 13, 2011
 ********************************************************************
 * Implementation of program A4_Control
 ********************************************************************)

PROGRAM _CYCLIC
VAR
    _p1 : BOOL;
    _e2 : R_TRIG;
    _e3 : R_TRIG;
    _e4 : R_TRIG;
    _e5 : F_TRIG;
    _e6 : F_TRIG;
END_VAR
(* Network 1: Enable Axis Request *)
_p1 := (NOT gA[4].Ind_Enabled OR gA[4].Cmd_Enable) AND gDriveSupply_Ready AND NOT gA[4].Error AND gA[4].Input_DriveEnable AND NOT gA[4].Cmd_EStopDisable;
gA[4].Cmd_Enable := _p1 AND ((NOT gA[7].Ind_Homing AND (g_iMachType = C_iRS15)) OR (g_iMachType = C_iRS26));

(* Network 2: Axis Ready For Operation *)
gA[4].Ind_Ready := gA[4].Ind_NetworkInit AND gA[4].Ind_ControllerReady AND gA[4].Ind_SynchronizedMotion;

(* Network 3: Axis Error Reset Request *)
_e2(CLK := gHMI_Reset_PB);
_e3(CLK := gA[4].Input_DriveEnable);
_e4(CLK := gCmd_ResetPBGen);
TOF_0(IN := _e2.Q OR _e3.Q OR _e4.Q, PT := T#20ms);
gA[4].Cmd_Reset := TOF_0.Q;

(* Network 4: Cam Automat Synchronization Permissive *)
Synch_Permissive := NOT gA[4].Error AND gA[4].Ind_Homed AND gA[4].Ind_Enabled AND gA[9].Ind_Homed AND NOT gA[4].Ind_Homing AND NOT gA[7].Ind_Homing;

(* Network 5: Cam Automat Synchronization Request *)
gA[4].Cmd_SynchronizedMotion := (NOT gA[4].Ind_AutomatEnabled OR gA[4].Cmd_SynchronizedMotion) AND Synch_Permissive AND NOT gRepeatChange AND NOT g_bChangeModTearingReq AND NOT g_bNumPliersChange4to2[1] AND NOT g_bNumPliersChange2to4[1];

(* Network 6: Advance/Retard Offset Trigger *)
TON_0(IN := gI_SS_TearingPos OR gI_SS_TearingNeg, PT := T#12ms);
HGW_Toggle_0(In := TON_0.Q, Time := T#12ms);

(* Network 7: Conversion offset increment from mm/bag to inch/bag *)
rIncrOffsetAxeRun_Inch := gr_rIncrOffsetAxeRun / 25.4;

(* Network 8: Advance Offset (+) *)
_e5(CLK := gA[4].Ind_bInContactZone);
IF gNever AND g_bMachineRun AND gManualMode_On AND gA[4].Ind_SynchronizedMotion AND gI_SS_TearingPos AND NOT gI_SS_TearingNeg AND _e5.Q THEN
    gRecipeActive.Tearing_Offset := gRecipeActive.Tearing_Offset + rIncrOffsetAxeRun_Inch;
END_IF;

(* Network 9: Offset Retard (-) *)
_e6(CLK := gA[4].Ind_bInContactZone);
IF gNever AND g_bMachineRun AND gManualMode_On AND gA[4].Ind_SynchronizedMotion AND gI_SS_TearingNeg AND NOT gI_SS_TearingPos AND _e6.Q THEN
    gRecipeActive.Tearing_Offset := gRecipeActive.Tearing_Offset + (rIncrOffsetAxeRun_Inch * -1.0);
END_IF;

(* Network 10: Limit The Offset To +/- The Active Repeat *)
gRecipeActive.Tearing_Offset := LIMIT(MN := gRecipeActive.Repeat * -1.0, IN := gRecipeActive.Tearing_Offset, MX := gRecipeActive.Repeat);

(* Network 11: Detect A Change In Offset And Trigger A Relative Change In Phase Offset *)
HGW_RelativeChangeReal1_0(IN_bEnable := g_bMachineRun, IN_rMax := gr_rLimOffsetRunVal, IN_rMin := gr_rLimOffsetRunVal * -1.0, IN_rInput := gRecipeActive.Holding_Offset, IN_rRepeat := gRecipeActive.Repeat, IN_rLimitIn := gRecipeActive.Tearing_Offset);
IF HGW_RelativeChangeReal1_0.OUT_bChange AND gA[4].Ind_SynchronizedMotion THEN
    gA[4].Cmd_PhaseOffset := TRUE;
END_IF;
gA[4].SP_PhaseOffset := HGW_RelativeChangeReal1_0.OUT_rDiff;
gRecipeActive.Tearing_Offset := HGW_RelativeChangeReal1_0.OUT_rLimitIn;

(* Network 12: Manu Axis motion timing setting (+) *)
gA[4].Cmd_ManuTimSetPlus := gManualMode_On AND NOT gA[9].Ind_InMotion AND NOT gMachine_Run AND NOT gMachine_Jog AND gI_SS_TearingPos AND NOT gI_SS_TearingNeg;

(* Network 13: Manu Axis motion timing setting (-) *)
gA[4].Cmd_ManuTimSetMinus := gManualMode_On AND NOT gA[9].Ind_InMotion AND NOT gMachine_Run AND NOT gMachine_Jog AND gI_SS_TearingNeg AND NOT gI_SS_TearingPos;

(* Network 14: Axis inside contact zone *)
gA[4].Ind_bInContactZone := gA[4].PositionDeg <= gr_rTearAxContactZone;
END_PROGRAM
```

#### A4_Control.var - Local variables
```iecst
(********************************************************************
 * COPYRIGHT -- Microsoft
 ********************************************************************
 * Program: A4_Control
 * File: A4_Control.var
 * Author: pkiel
 * Created: July 13, 2011
 ********************************************************************
 * Local variables of program A4_Control
 ********************************************************************)
VAR
	HGW_ChangeReal_0 : HGW_ChangeReal;
	HGW_RelativeChangeReal1_0 : H_FB_RelativeChangeLimitReal1;
	HGW_Toggle_0 : HGW_Toggle;
	Synch_Permissive : BOOL;
	TOF_0 : TOF;
	TON_0 : TON;
  rIncrOffsetAxeRun_Inch : REAL ;
END_VAR
```

### Program Logical/BagMachine_Section/Tearing/Axis4/A4_Automat (IEC) - Cam Automat

#### A4_Automat.var
```iecst
(********************************************************************
 * COPYRIGHT -- Microsoft
 ********************************************************************
 * Program: A4_Automat
 * File: A4_Automat.var
 * Author: pkiel
 * Created: July 13, 2011
 ********************************************************************
 * Local variables of program A4_Automat
 ********************************************************************)
VAR
	AutData : MC_AUTDATA_TYP;
	AutomatStart : BOOL;
	ErrorID : UINT;
	MasterOffset : REAL;
  MasterParID : UINT;
  uiMasterParID1 : UINT;
  uiSP_MasterParID : UINT;
  uiiSP_Master : UDINT;
  bCmdSynchroOn : BOOL ;
  bCmdSynchroOff : BOOL ;
  bCmdSynchroOn1 : BOOL ;
  bCmdSynchroOff1 : BOOL ;
  uiiSP_MasterFactor : UDINT ;
  uiiSP_SlaveFactor : UDINT ;
	MC_BR_AutControl_0 : MC_BR_AutControl;
  uiMC_BR_AutControl_0_MemoErrorID : UINT ;
  MC_BR_InitMasterParIDTransfer_0 : MC_BR_InitMasterParIDTransfer;
  MC_BR_InitMasterParIDTransfer_1 : MC_BR_InitMasterParIDTransfer;
  ParID_Ready : BOOL;
  ParID_Ready1 : BOOL;
	PositionMOD : DINT;
	PositionOffset : DINT;
	SlaveStartOffset : REAL;
	Synch_Request : BOOL;
  bTest_ : ARRAY[0..9] OF  BOOL;
  iTest_ : ARRAY[0..9] OF  INT;
  rTest_ : ARRAY[0..9] OF  REAL;
  rMaCompDist : REAL ;
  rSPMaPos    : REAL ;
  rOffsetDeg  : REAL ;
  rSlCompDist : REAL ;
  rTemp_      : ARRAY[0..9] OF REAL ;
  usiMemoStat : USINT;
  iIndex : INT ;
  rMaCompDistStat6 : REAL;
  rSlCompDistStat6 : REAL;
  rMasterFactor5 : REAL;
  iiMasterFactor5 : DINT;
  iiSlaveFactor5  : DINT;
  rSlave_AxisPeriod : REAL ;
END_VAR
```

#### A4_AutomatCyclic.st
```iecst
(********************************************************************
 * COPYRIGHT -- Microsoft
 ********************************************************************
 * Program: A4_Automat
 * File: A4_AutomatCyclic.st
 * Author: pkiel
 * Created: July 13, 2011
 ********************************************************************
 * Implementation of program A4_Automat
 ********************************************************************)

PROGRAM _CYCLIC

      // Synchro ratio Master/Slave
      iIndex := MC_BR_AutControl_0.ActualStateIndex ;
      CASE iIndex OF
        3 : // Master = Holding
            //gA[4].rRSynNum := 2.0 ;        D.M. 03/02/2012 Pyrollpack_14661 Suppress cause is not correct for offset Virtual Masrter / Slave calculation in A4_Basic and not used in setting mode Automat states 3 and 4
            //gA[4].rRSynDen := 1.0 ;
        4 : // Master = Holding
            //gA[4].rRSynNum := 4.0 ;
            //gA[4].rRSynDen := 1.0 ;
      ELSE  // Master = Virtual
            IF (g_rNumbPliers <> 0.0) THEN
              gA[4].rRSynNum := 4.0 / g_rNumbPliers ;
            ELSE
              gA[4].rRSynNum := 1.0 ;
            END_IF
            gA[4].rRSynDen := 1.0 ;
      END_CASE

(**** STRAIGHT GEARED CAM AUTOMAT WITH ABSOLUTE PHASE SYNCHRONIZATION FOR TEARING AXIS ***)

(* Set Up Master Position Parameter ID *)

  // Maintaining+Tearing+Drum timing setting
  IF gstCycA[3].CycManTimSet.CmdSynchroOn THEN
    IF gA[3].rRSynDen < 4 THEN
      MC_BR_AutControl_0.Signal1 := 1 ;
    ELSIF gA[3].rRSynDen >= 4 THEN
      MC_BR_AutControl_0.Signal2 := 1 ;
    END_IF
    MC_BR_AutControl_0.Signal3 := 0 ;
  ELSE
    MC_BR_AutControl_0.Signal1 := 0 ;
    MC_BR_AutControl_0.Signal2 := 0 ;
    MC_BR_AutControl_0.Signal3 := 1 ;
  END_IF

  // A4 Synchro OK indicator
  gstCycA[3].CycManTimSet.bSynchroOkSlavA[4] := ( MC_BR_InitMasterParIDTransfer_1.Master = gA[3].Ident )                                AND
                                                ( MC_BR_InitMasterParIDTransfer_1.MasterParID = gstCycA[3].CycManTimSet.uiMasterParID ) AND
                                                ( MC_BR_AutControl_0.ActualStateIndex = 3 OR MC_BR_AutControl_0.ActualStateIndex = 4 )  AND
                                                gA[4].Ind_SynchronizedMotion AND ParID_Ready ;

  // Tearing+Drum timing setting
  IF gstCycA[4].CycManTimSet.bCyc THEN
    IF (gstCycA[4].CycManTimSet.CmdSynchroOn) THEN
      MC_BR_AutControl_0.Signal1 := 0 ;
      MC_BR_AutControl_0.Signal2 := 0 ;
      MC_BR_AutControl_0.Signal3 := 1 ;
    ELSE
      MC_BR_AutControl_0.Signal1 := 0 ;
      MC_BR_AutControl_0.Signal2 := 0 ;
      MC_BR_AutControl_0.Signal3 := 0 ;
    END_IF
  END_IF

  IF gstCycA[3].CycManTimSet.bFCyc AND
     gstCycA[4].CycManTimSet.bFCyc THEN
    MC_BR_AutControl_0.Signal1 := 0 ;
    MC_BR_AutControl_0.Signal2 := 0 ;
    MC_BR_AutControl_0.Signal3 := 0 ;
  END_IF

  // A4 Synchro OK indicator
  gstCycA[4].CycManTimSet.bSynchroOkSlavA[4] := ( MC_BR_AutControl_0.ActualStateIndex = 2 )  AND
                                                gA[4].Ind_SynchronizedMotion AND ParID_Ready ;

  //Synch_Request := gA[4].Cmd_SynchronizedMotion ;
  Synch_Request := gA[4].Cmd_SynchronizedMotion AND NOT(MC_BR_AutControl_0.Stop) ;  // D.M. 26/01/2012 RS26 Pyrollpack_14661 added because it happened that Stop=1 and Synch_Request=1 => MC_BR_AutControl_0 makes fault 29256
	IF (Synch_Request AND NOT ParID_Ready) THEN
    MC_BR_InitMasterParIDTransfer_0.Master:= gA[9].Ident ;
    MC_BR_InitMasterParIDTransfer_0.Slave:=gA[4].Ident;
    MC_BR_InitMasterParIDTransfer_0.MasterParID:= 412 ; // ParID 412 = VAX Position (in case virtual axis)
    MC_BR_InitMasterParIDTransfer_0.SlaveChannel:=0;
    MC_BR_InitMasterParIDTransfer_0.Execute:= 1 ;
    IF (MC_BR_InitMasterParIDTransfer_0.Done) THEN
      MasterParID:=MC_BR_InitMasterParIDTransfer_0.ReceiveParID;
      MC_BR_InitMasterParIDTransfer_0.Execute:=FALSE;
      ParID_Ready1:=1;
    ELSIF (MC_BR_InitMasterParIDTransfer_0.Error) THEN
    (*Store ErrorID in a variable,
      ErrorID is reset on falling edge of 'Execute'*)
      ErrorID:=MC_BR_InitMasterParIDTransfer_0.ErrorID;
      ParID_Ready1:=0;
      MC_BR_InitMasterParIDTransfer_0.Execute:=FALSE;
    END_IF
    MC_BR_InitMasterParIDTransfer_1.Master       := gA[3].Ident ;
    MC_BR_InitMasterParIDTransfer_1.Slave        := gA[4].Ident;
    MC_BR_InitMasterParIDTransfer_1.MasterParID  := gstCycA[3].CycManTimSet.uiMasterParID ;
    MC_BR_InitMasterParIDTransfer_1.SlaveChannel := 2 ;
    MC_BR_InitMasterParIDTransfer_1.Execute      := 1 ;
    IF (MC_BR_InitMasterParIDTransfer_1.Done) AND ParID_Ready1 THEN
      uiMasterParID1:=MC_BR_InitMasterParIDTransfer_1.ReceiveParID;
      MC_BR_InitMasterParIDTransfer_1.Execute:=FALSE;
      ParID_Ready:=1;
    ELSIF (MC_BR_InitMasterParIDTransfer_1.Error) THEN
    (*Store ErrorID in a variable,
      ErrorID is reset on falling edge of 'Execute'*)
      ErrorID:=MC_BR_InitMasterParIDTransfer_1.ErrorID;
      ParID_Ready:=0;
      MC_BR_InitMasterParIDTransfer_1.Execute:=FALSE;
    END_IF
	END_IF
  MC_BR_InitMasterParIDTransfer_0();
  MC_BR_InitMasterParIDTransfer_1();

(**** Initialize Automat Parameters Upon Automat Start Request ****)
	IF (EDGEPOS(ParID_Ready))THEN

		(**** Calculate Slave Start Offset ****)
			MasterOffset := gRecipeActive.Tearing_Offset+gRecipeActive.Holding_Offset;
			PositionOffset:= REAL_TO_DINT((gA[9].PositionInch-(gA[4].PositionInch-MasterOffset))*1000);
			PositionMOD:= REAL_TO_DINT(gRecipeActive.Repeat*1000);
			SlaveStartOffset:= (DINT_TO_REAL(PositionOffset MOD PositionMOD))/1000;
			IF (SlaveStartOffset >= (0.5*gRecipeActive.Repeat)) THEN
				SlaveStartOffset := SlaveStartOffset - gRecipeActive.Repeat;
			END_IF
			IF (SlaveStartOffset < (-0.5*gRecipeActive.Repeat)) THEN
				SlaveStartOffset := SlaveStartOffset + gRecipeActive.Repeat;
			END_IF

      rSlave_AxisPeriod := gA[4].AxisPeriod * gA[4].rRSynNum/gA[4].rRSynDen ;
      rOffsetDeg := gRecipeActive.rTearing_PhasMasterDeg ;

      rSPMaPos := (gA[4].PositionDeg - rOffsetDeg)/(gA[4].rRSynNum/gA[4].rRSynDen) ;
      rTemp_[0] := rSPMaPos - gA[9].PositionDeg ;
      rMaCompDist := H_FC_Modulus (
                          IN_rMod := (360 * gA[4].rRSynNum/gA[4].rRSynDen) ,
                          IN_rVar := rTemp_[0]
                                  ) ;

		(*general automat parameter*)
			//AutData.Master				    := gA[3].Ident;
			AutData.MasterParID			  := MasterParID;
			AutData.StartPosition		  := 0;
			AutData.StartInterval		  := gA[9].AxisPeriod;
			AutData.MaxMasterVelocity	:= gr_rMachMaxSpeed_BPM ;

		//Automat STATE 0 Basis State
			AutData.State[0].Event[0].Type		  := ncST_END;
			AutData.State[0].Event[0].Attribute	:= ncAT_ONCE;
      IF gA[4].Ind_bInContactZone                  AND
         (g_iMachType = C_iRS15)                   AND
         NOT(gstCycA[3].CycManTimSet.CmdSynchroOn) AND
         NOT(gstCycA[4].CycManTimSet.CmdSynchroOn) THEN
        // Start synchro with tearing in contact zone
        AutData.State[0].Event[0].NextState := 5;
      ELSIF (rMaCompDist >= 1/gA[9].UnitsPerDeg) AND // rMaCompDist must be >= 1 Units
            gA[4].bSynchroReq                    THEN
		  	AutData.State[0].Event[0].NextState	:= 1;
      ELSE
        rMaCompDist := 1/gA[9].UnitsPerDeg ;
        AutData.State[0].Event[0].NextState := 2;
      END_IF

    //Automat STATE 1 Master/Slave Absolute Phase Correction
      AutData.State[1].MasterParID        := MasterParID;
      AutData.State[1].CamProfileIndex    := 16#FFFF;
      AutData.State[1].MasterFactor       := REAL_TO_UDINT(rMaCompDist * gA[4].UnitsPerDeg) ;
      AutData.State[1].SlaveFactor        := 0 ;
      AutData.State[1].CompMode           := ncOFF;

      AutData.State[1].Event[0].Type      := ncST_END ;
      AutData.State[1].Event[0].Attribute := ncST_END ;
      AutData.State[1].Event[0].NextState := 2 ;

      AutData.State[1].Event[1].Type      := ncSIGNAL1 ;
      AutData.State[1].Event[1].Attribute := ncAT_ONCE ;
      AutData.State[1].Event[1].NextState := 3 ;

      AutData.State[1].Event[2].Type      := ncSIGNAL2;
      AutData.State[1].Event[2].Attribute := ncAT_ONCE;
      AutData.State[1].Event[2].NextState := 4;

      AutData.State[1].Event[3].Type      := ncSIGNAL3;
      AutData.State[1].Event[3].Attribute := ncAT_ONCE;
      AutData.State[1].Event[3].NextState := 2;

    //Automat STATE 2 Master/Slave run
      AutData.State[2].MasterParID     := MasterParID;
      AutData.State[2].CamProfileIndex := 16#FFFF;
      AutData.State[2].MasterFactor    := REAL_TO_UDINT(gA[9].AxisPeriod);
      AutData.State[2].SlaveFactor     := REAL_TO_UDINT(rSlave_AxisPeriod);
      AutData.State[2].CompMode        := ncOFF;

      AutData.State[2].Event[0].Type      := ncST_END ;
      AutData.State[2].Event[0].Attribute := ncST_END;
      AutData.State[2].Event[0].NextState := 2;

      AutData.State[2].Event[1].Type      := ncST_END+ncNEGATIVE ;
      AutData.State[2].Event[1].Attribute := ncST_END;
      AutData.State[2].Event[1].NextState := 2;

      AutData.State[2].Event[2].Type      := ncSIGNAL1;
      AutData.State[2].Event[2].Attribute := ncAT_ONCE;
      AutData.State[2].Event[2].NextState := 3;

      AutData.State[2].Event[3].Type      := ncSIGNAL2;
      AutData.State[2].Event[3].Attribute := ncAT_ONCE;
      AutData.State[2].Event[3].NextState := 4;

    //Automat STATE 3 Master/Slave Timing setting case 1
      AutData.State[3].MasterParID     := uiMasterParID1;
      AutData.State[3].CamProfileIndex := 16#FFFF;
      AutData.State[3].MasterFactor    := REAL_TO_UDINT(gA[3].AxisPeriod);
      AutData.State[3].SlaveFactor     := REAL_TO_UDINT(gA[4].AxisPeriod*2);
      AutData.State[3].CompMode        := ncOFF;

      AutData.State[3].Event[0].Type       := ncST_END ;
      AutData.State[3].Event[0].Attribute  := ncST_END ;
      AutData.State[3].Event[0].NextState  := 3 ;

      AutData.State[3].Event[1].Type       := ncST_END+ncNEGATIVE ;
      AutData.State[3].Event[1].Attribute  := ncST_END ;
      AutData.State[3].Event[1].NextState  := 3 ;

      AutData.State[3].Event[2].Type       := ncSIGNAL3 ;
      AutData.State[3].Event[2].Attribute  := ncAT_ONCE ;
      AutData.State[3].Event[2].NextState  := 2 ;

    //Automat STATE 4 Master/Slave Timing setting case 2
      AutData.State[4].MasterParID     := uiMasterParID1;
      AutData.State[4].CamProfileIndex := 16#FFFF;
      AutData.State[4].MasterFactor    := REAL_TO_UDINT(gA[3].AxisPeriod);
      AutData.State[4].SlaveFactor     := REAL_TO_UDINT(gA[4].AxisPeriod*4);
      AutData.State[4].CompMode        := ncOFF;

      AutData.State[4].Event[0].Type       := ncST_END ;
      AutData.State[4].Event[0].Attribute  := ncST_END ;
      AutData.State[4].Event[0].NextState  := 4 ;

      AutData.State[4].Event[1].Type       := ncST_END+ncNEGATIVE ;
      AutData.State[4].Event[1].Attribute  := ncST_END ;
      AutData.State[4].Event[1].NextState  := 4 ;

      AutData.State[4].Event[2].Type       := ncSIGNAL3 ;
      AutData.State[4].Event[2].Attribute  := ncAT_ONCE ;
      AutData.State[4].Event[2].NextState  := 2 ;

			MC_BR_AutControl_0.Enable 		  := 1;
			MC_BR_AutControl_0.AdrAutData 	:= ADR(AutData);
			MC_BR_AutControl_0.InitAutData 	:= 1;

    //Automat STATE 5 Master/Slave
      iiMasterFactor5 := REAL_TO_UDINT(rMaCompDist*gA[9].UnitsPerDeg) ;
      IF iiMasterFactor5 < 1 THEN
        iiMasterFactor5 := REAL_TO_UDINT(gA[9].AxisPeriod) ;
        iiSlaveFactor5  := REAL_TO_UDINT(gA[4].AxisPeriod) ;
      ELSE
        iiSlaveFactor5 := 0 ;
      END_IF ;
      AutData.State[5].MasterParID     := MasterParID;
      AutData.State[5].CamProfileIndex := 16#FFFF;
      AutData.State[5].MasterFactor    := iiMasterFactor5 ;
      AutData.State[5].SlaveFactor     := iiSlaveFactor5 ;
      AutData.State[5].CompMode        := ncOFF;

      AutData.State[5].Event[0].Type       := ncST_END ;
      AutData.State[5].Event[0].Attribute  := ncST_END ;
      AutData.State[5].Event[0].NextState  := 2 ;

      AutData.State[5].Event[2].Type      := ncSIGNAL1;
      AutData.State[5].Event[2].Attribute := ncAT_ONCE;
      AutData.State[5].Event[2].NextState := 3;

      AutData.State[5].Event[3].Type      := ncSIGNAL2;
      AutData.State[5].Event[3].Attribute := ncAT_ONCE;
      AutData.State[5].Event[3].NextState := 4;

      AutData.State[5].Event[3].Type      := ncSIGNAL3;
      AutData.State[5].Event[3].Attribute := ncAT_ONCE;
      AutData.State[5].Event[3].NextState := 2;

      MC_BR_AutControl_0.Enable      := 1;
      MC_BR_AutControl_0.AdrAutData  := ADR(AutData);
      MC_BR_AutControl_0.InitAutData := 1;
  END_IF

			(* wait for initialization done or restart *)
			IF ((MC_BR_AutControl_0.AutDataInitialized=1) AND (Synch_Request)) THEN
				MC_BR_AutControl_0.InitAutData := 0;
				MC_BR_AutControl_0.Enable :=1;
				AutomatStart := 1;
        uiMC_BR_AutControl_0_MemoErrorID := 0 ;
			END_IF
			(* check if error occured *)
			IF (MC_BR_AutControl_0.ErrorID <> 0) THEN
        uiMC_BR_AutControl_0_MemoErrorID := MC_BR_AutControl_0.ErrorID ;
				MC_BR_AutControl_0.Enable := 0;
			END_IF

	(******************** ENABLE CAM-AUTOMAT **********************)

	IF (AutomatStart) THEN
			MC_BR_AutControl_0.Start := 1;
			AutomatStart := 0;
	END_IF

	IF (NOT Synch_Request) THEN
			MC_BR_AutControl_0.Stop := 1;
			MC_BR_AutControl_0.Start := 0;
      ParID_Ready := 0;
      ParID_Ready1 := 0;
			IF (MC_BR_AutControl_0.Running=0) THEN
				MC_BR_AutControl_0.Enable := 0;
				MC_BR_AutControl_0.Stop := 0;
			END_IF
   //*************************************************
   // D.M. 26/01/2012 RS26 Pyrollpack_14661 added because after guard fault it happened that Stop=1 and MC_BR_AutControl_0.Enable => not possible to finish MC_BR_AutControl_0 => program locked
      IF MC_BR_AutControl_0.Stop        AND
         NOT(MC_BR_AutControl_0.Enable) THEN
        MC_BR_AutControl_0.Enable := 1 ;
      END_IF
   //*************************************************
  END_IF

	gA[4].Ind_AutomatEnabled:=MC_BR_AutControl_0.Enable;
	gA[4].Ind_CurrentAutomatState:=MC_BR_AutControl_0.ActualStateIndex;
  gA[4].Ind_bSynchroOK := (MC_BR_AutControl_0.ActualStateIndex >= 2) AND gA[4].Ind_SynchronizedMotion ; ;

	(********************** MC_AUTCONTROL *************************)
	MC_BR_AutControl_0.Slave:= gA[4].Ident;
	MC_BR_AutControl_0();

END_PROGRAM
```

### Program Logical/BagMachine_Section/Tearing/Axis4/A4_Cycle (IEC) - A new program

#### A4_CycleCyclic.st
```iecst
(********************************************************************
 * COPYRIGHT -- .
 ********************************************************************
 * Program: A1_Cycle
 * File: A1_CycleCyclic.st
 * Author: dominique
 * Created: August 01, 2011
 ********************************************************************
 * Implementation of program A1_Cycle
 ********************************************************************)

PROGRAM _CYCLIC

// Manu axis movement for timing setting

    //---------------------------------------------------------------------------------------------------------------------
    // Tearing timing setting cycle
    //---------------------------------------------------------------------------------------------------------------------
    // Start cycle
    gstCycA[4].CycManTimSet.CmdStart := ( gA[4].Cmd_ManuTimSetPlus        OR
                                          gA[4].Cmd_ManuTimSetMinus )     AND
                                        ( NOT(g_bCycManTimeSetOn)         OR
                                          gstCycA[4].CycManTimSet.bSCyc ) AND
                                        gA[4].Ind_Ready                   AND
                                        gA[7].Ind_Ready                   ;
    IF gstCycA[4].CycManTimSet.CmdStart THEN
      gstCycA[4].CycManTimSet.bSCyc := 1 ;
    END_IF ;

    //----------------------------------------------------------------------
    // Cycle at rest
    IF NOT(gstCycA[4].CycManTimSet.bSCyc) AND
       1                                 THEN
      IF NOT( gstCycA[4].CycManTimSet.bFCyc ) THEN
        // Init after cycle unpropaly ended
        gstCycA[4].CycManTimSet.bFCyc := 1 ;
        gstCycA[4].CycManTimSet.bCyc  := 0 ;

        gstCycA[4].CycManTimSet.CmdMov       := 0 ;
        gstCycA[4].CycManTimSet.CmdStop      := 0 ;
        gstCycA[4].CycManTimSet.CmdSynchroOn := 0 ;

        gA[4].Cmd_Override  := 1 ;
        gA[4].rSP_OverrideA := 1.0 ;
      END_IF
      gstCycA[4].CycManTimSet.iStep := 0 ;
      RETURN ;
    ELSE
    //----------------------------------------------------------------------
    // Cycle running

      // Permanent conditions
      IF NOT(gA[4].Ind_Ready)                  OR
         NOT(gA[7].Ind_Ready)                  OR
         NOT(gstCycA[4].CycManTimSet.CmdStart) AND
         (gstCycA[4].CycManTimSet.iStep <= 2)  THEN
        gstCycA[4].CycManTimSet.bSCyc := 0 ;
        RETURN ;
      END_IF

      // Permanent actions
      stTON_01 (
            IN := ( gstCycA[4].CycManTimSet.iStep = C_iSTEP_0 ) ,
            PT := T#30ms
               ) ;

      // Phasing override acce management
      IF EDGEPOS(gstCycA[4].CycManTimSet.CmdStart) THEN
        IF gstCycA[4].CycManTimSet.CmdStart THEN
          gA[4].rSP_OverrideA := 0.5 ;
          iTest_[0] := iTest_[0] + 1 ;
        ELSE
          gA[4].rSP_OverrideA := 1.0 ;
          iTest_[1] := iTest_[1] + 1 ;
        END_IF
        iTest_[2] := iTest_[2] + 1 ;
        gA[4].Cmd_Override := 1 ;
      END_IF

    END_IF
    //----------------------------------------------------------------------
    // Cycle steps

        CASE gstCycA[4].CycManTimSet.iStep OF

        C_iSTEP_0 :
         //----------------------------------------------
         // Etape 1 : Initialisation
         //----------------------------------------------
          IF stTON_01.Q THEN
            gstCycA[4].CycManTimSet.iStep := C_iSTEP_1 ;

            // Action Step 1
            gstCycA[4].CycManTimSet.bFCyc := 0 ;
            gstCycA[4].CycManTimSet.bCyc  := 1 ;
          END_IF

        C_iSTEP_1 :
         //----------------------------------------------
         // Etape 2 : Synchro Drum on Tearing
         //----------------------------------------------
          IF TRUE THEN
            gstCycA[4].CycManTimSet.iStep := C_iSTEP_2 ;

            // Action Step 2
            gstCycA[4].CycManTimSet.CmdSynchroOn := 1 ;
            gA[4].Cmd_Override := 1 ;
          END_IF

        C_iSTEP_2 :
         //----------------------------------------------
         // Step 3 : Activation motion and Stop waiting
         //----------------------------------------------
          IF gstCycA[4].CycManTimSet.bSynchroOkSlavA[4]    AND
             gstCycA[4].CycManTimSet.bSynchroOkSlavA[7]    AND
             ( gstCycA[4].CycManTimSet.bSynchroOkSlavA[12] OR
               NOT(gA[12].bInMach) )                       AND
             ( gstCycA[4].CycManTimSet.bSynchroOkSlavA[13] OR
               NOT(gA[13].bInMach) )                       THEN
            gstCycA[4].CycManTimSet.iStep := C_iSTEP_3 ;

            // Action Step 3
            gstCycA[4].CycManTimSet.CmdMov  := 1 ;
            gstCycA[4].CycManTimSet.CmdStop := 0 ;
            // Stop waiting
          END_IF

        C_iSTEP_3 :
         //----------------------------------------------
         // Step 4 : Stop motion and End stop waiting
         //----------------------------------------------
          IF NOT(gstCycA[4].CycManTimSet.CmdStart) THEN
            gstCycA[4].CycManTimSet.iStep := C_iSTEP_4 ;

            // Action Step 4
            gstCycA[4].CycManTimSet.CmdMov  := 0 ;
            gstCycA[4].CycManTimSet.CmdStop := 1 ;
            // End stop waiting
          END_IF

        C_iSTEP_4 :
         //----------------------------------------------
         // Step 3 : Activation motion and Stop waiting
         // Step 5 : Cut synchro
         //----------------------------------------------
          // Condition Step3
          IF gstCycA[4].CycManTimSet.CmdStart THEN
            gstCycA[4].CycManTimSet.iStep := C_iSTEP_3 ;

            // Action Step 3
            gstCycA[4].CycManTimSet.CmdMov  := 1 ;
            gstCycA[4].CycManTimSet.CmdStop := 0 ;
            // Stop waiting
            RETURN ;
          END_IF ;
          // Condition Step5
          IF NOT(gstCycA[4].CycManTimSet.CmdStop) THEN
            gstCycA[4].CycManTimSet.iStep := C_iSTEP_5 ;

            // Action Step 5
            gstCycA[4].CycManTimSet.CmdSynchroOn := 0 ;
          END_IF

        C_iSTEP_5 :
         //----------------------------------------------
         // Step 6 : New offset calculation
         //----------------------------------------------
          IF NOT(gstCycA[4].CycManTimSet.bSynchroOkSlavA[7])    AND
             ( NOT(gstCycA[4].CycManTimSet.bSynchroOkSlavA[12]) OR
               NOT(gA[12].bInMach) )                            AND
             ( NOT(gstCycA[4].CycManTimSet.bSynchroOkSlavA[13]) OR
               NOT(gA[13].bInMach) )                            THEN
            gstCycA[4].CycManTimSet.iStep := C_iSTEP_6 ;

            // Action Step 6
            // Memo Actual phase Offset
            rTempActPhasDeg[4] := gRecipeActive.rTearing_PhasMasterDeg ;
            rTempActOffsetInch[4] := gRecipeActive.Tearing_Offset ;
            // Update phase
            gRecipeActive.rTearing_PhasMasterDeg := gA[4].rActPhasDeg ;
            gRecipeActive.rDrum_PhasMasterDeg    := gA[7].rActPhasDeg ;
            IF gA[12].bInMach THEN
              gRecipeActive.rEnvB_PhasMasterDeg := gA[12].rActPhasDeg ;
            END_IF
            IF gA[13].bInMach THEN
              gRecipeActive.rTearEB_PhasMasterDeg := gA[13].rActPhasDeg ;
            END_IF
            // Update Offset
            rTemp_[4] := rTempActOffsetInch[4] + (gRecipeActive.rTearing_PhasMasterDeg - rTempActPhasDeg[4])/(gA[4].rRSynNum/gA[4].rRSynDen)*gA[4].InchPerDeg ;
            gRecipeActive.Tearing_Offset := H_FC_Modulus (IN_rMod := gRecipeActive.Repeat, IN_rVar := rTemp_[4]) ;
          END_IF

        C_iSTEP_6 :
         //----------------------------------------------
         // Step 0 : First step
         //----------------------------------------------
          IF NOT(gstCycA[4].CycManTimSet.bSynchroOkSlavA[7])    AND
             ( NOT(gstCycA[4].CycManTimSet.bSynchroOkSlavA[12]) OR
               NOT(gA[12].bInMach) )                            AND
             ( NOT(gstCycA[4].CycManTimSet.bSynchroOkSlavA[13]) OR
               NOT(gA[13].bInMach) )                            AND
             (gA[4].Ind_CurrentAutomatState <> 3)               THEN
            gstCycA[4].CycManTimSet.iStep := C_iSTEP_0 ;

            // Action Step 0
            gstCycA[4].CycManTimSet.bSCyc := 0 ;
            gstCycA[4].CycManTimSet.bFCyc := 1 ;
            gstCycA[4].CycManTimSet.bCyc  := 0 ;
          END_IF
        END_CASE
    //---------------------------------------------------------------------------------------------------------------------

END_PROGRAM
```

#### A4_CycleInit.st
```iecst
(********************************************************************
 * COPYRIGHT -- .
 ********************************************************************
 * Program: A1_Cycle
 * File: A1_CycleInit.st
 * Author: dominique
 * Created: August 01, 2011
 ********************************************************************
 * Implementation of program A1_Cycle
 ********************************************************************)

PROGRAM _INIT

  gstCycA[4].CycManTimSet.uiMasterParID := 428 ; // ParID 428 = CTRL Position controller: Input set position (in case real axis)

END_PROGRAM
```

### Package Logical/BagMachine_Section/EntryPull - Axis

- Program Logical/BagMachine_Section/EntryPull/EntryNip (IEC) - Entry Air Nip Control (no source held here)

### Data object Logical/BagMachine_Section/EntryPull/Axis5/A5_Par (Apt) - Servo Axis Parameter File

#### A5_Par.apt
```
AcoposParameterTable:
  Root Parameters:
    110 = ncSW_OFF (Name=CMD_SIMULATION)  // Simulation mode: Command
    128 = 1 (Name=SGEN_SW_END_IGNORE)  // SGEN_SW_END_IGNORE
```

### Program Logical/BagMachine_Section/EntryPull/Axis5/A5_Basic (IEC) - Basic Servo

#### A5_BasicCyclic.st - Cyclic code
```iecst
(********************************************************************
 * COPYRIGHT -- Microsoft
 ********************************************************************
 * Program: A5_Basic
 * File: A5_BasicCyclic.st
 * Author: pkiel
 * Created: July 13, 2011
 ********************************************************************
 * Implementation of program A5_Basic
 ********************************************************************)

PROGRAM _CYCLIC

	IF (gA[5].Ident<>0) THEN

	(************************ READ DRIVE STATUS *************************)
	(* Access to the following bools:
	gA[x]_DriveStatus.Simulation			: If TRUE, simulation mode is active
	gA[x]_DriveStatus.NetworkInit			: If TRUE, the network is initialized
	gA[x]_DriveStatus.HomeSwitch			: If TRUE, the digital reference switch input is active
	gA[x]_DriveStatus.PosHWSwitch			: If TRUE, the positive hardware end switch is active
	gA[x]_DriveStatus.NegHWSwitch			: If TRUE, the negative hardware end switch is active
	gA[x]_DriveStatus.Trigger1				: If TRUE, the first trigger input is active
	gA[x]_DriveStatus.Trigger2				: If TRUE, the second trigger input is active
	gA[x]_DriveStatus.DriveEnable			: If TRUE, the enable input is active
	gA[x]_DriveStatus.ControllerReady		: If TRUE, the controller is ready to beturned on
	gA[x]_DriveStatus.ControllerStatus		: If TRUE, the controller is turned on (Same as MC_Power.Status)
	gA[x]_DriveStatus.AxisError				: If TRUE, at least one error has occurred (not acknowledged)
	gA[x]_DriveStatus.LagWarning			: If TRUE, the lag error has exceeded the limit value specified for a warning*)
		MC_BR_ReadDriveStatus_0.Enable := 1;
		MC_BR_ReadDriveStatus_0.Axis := gA[5].Ident;
		MC_BR_ReadDriveStatus_0.AdrDriveStatus := ADR (DriveStatus);
		MC_BR_ReadDriveStatus_0();
		gA[5].Ind_Simulation		:=	DriveStatus.Simulation;
		gA[5].Ind_NetworkInit		:=	DriveStatus.NetworkInit;
		gA[5].Input_Home			:=	DriveStatus.HomeSwitch;
		gA[5].Input_PosHW			:=	DriveStatus.PosHWSwitch;
		gA[5].Input_NegHW			:=	DriveStatus.NegHWSwitch;
		gA[5].Input_Trigger1		:=	DriveStatus.Trigger1;
		gA[5].Input_Trigger2		:=	DriveStatus.Trigger2;
		gA[5].Input_DriveEnable		:=	DriveStatus.DriveEnable;
		gA[5].Ind_ControllerReady	:=	DriveStatus.ControllerReady;
		gA[5].Ind_ControllerStatus	:=	DriveStatus.ControllerStatus;
		gA[5].Error					:=	DriveStatus.AxisError;
		gA[5].Ind_LagWarning		:=	DriveStatus.LagWarning;

	(************************ READ AXIS ERROR **********************)
		MC_ReadAxisError_0.Enable := gA[5].Ind_NetworkInit;
		MC_ReadAxisError_0.Axis := gA[5].Ident;
		MC_ReadAxisError_0.DataAddress := ADR(gA[5].ErrorText);
		MC_ReadAxisError_0.DataLength := SIZEOF(gA[5].ErrorText);
		MC_ReadAxisError_0.DataObjectName := 'Error_Eng';
		MC_ReadAxisError_0();
		IF(MC_ReadAxisError_0.Valid) THEN
			gA[5].ErrorID := MC_ReadAxisError_0.AxisErrorID;
			gA[5].ErrorCount := MC_ReadAxisError_0.AxisErrorCount;
		END_IF
	(* Auto Acknowledge Errors *)
		IF (gA[5].Cmd_Reset AND (gA[5].ErrorCount<>0) AND NOT AutoAck) THEN
			AutoAck:=1;
		ELSE
			AutoAck:=0;
		END_IF
	(*Axis Error Acknowledge*)
		IF (EDGEPOS(AutoAck) OR EDGEPOS(gA[5].ErrorAck)) THEN
			MC_ReadAxisError_0.Acknowledge := 1;
		ELSE;
			MC_ReadAxisError_0.Acknowledge :=0;
		END_IF

	(************************ RESET AXIS ERROR **********************)
		IF (gA[5].Cmd_Reset AND (gA[5].ErrorCount=0) AND gA[5].ErrorStop) THEN
			MC_Reset_0.Execute:=1;
		END_IF
		IF (MC_Reset_0.Done) THEN
			MC_Reset_0.Execute:=0;
			gA[5].Cmd_Reset:=0;
			ResetError := 0;
		END_IF
		IF (MC_Reset_0.Error) THEN
			MC_Reset_0.Execute:=0;
			gA[5].Cmd_Reset:=0;
			ResetError := 1;
		END_IF
		MC_Reset_0.Axis:=gA[5].Ident;
		MC_Reset_0();

	(************************ READ AXIS STATUS *************************)
		MC_ReadStatus_0.Enable := gA[5].Ind_NetworkInit;
		MC_ReadStatus_0.Axis := gA[5].Ident;
		MC_ReadStatus_0();
		IF(MC_ReadStatus_0.Valid = TRUE)THEN
			gA[5].Ind_Enabled 			:= NOT (MC_ReadStatus_0.Disabled);
			gA[5].Ind_StandStill		:= MC_ReadStatus_0.StandStill;
			gA[5].Ind_Stopping			:= MC_ReadStatus_0.Stopping;
			gA[5].Ind_DiscreteMotion	:= MC_ReadStatus_0.DiscreteMotion;
			gA[5].Ind_ContinuousMotion	:= MC_ReadStatus_0.ContinuousMotion;
			gA[5].Ind_SynchronizedMotion:= MC_ReadStatus_0.SynchronizedMotion;
			gA[5].ErrorStop				:= MC_ReadStatus_0.Errorstop;
		END_IF

	(******************** INIT POSITION MODULUS  *********************)
		MC_BR_InitModPos_0.Execute:= InitModPosition;
		MC_BR_InitModPos_0.Axis:= gA[5].Ident;
		MC_BR_InitModPos_0.Period:= REAL_TO_UDINT(gA[5].AxisPeriod);
		MC_BR_InitModPos_0.Factor:=1;
		InitModPos_Done:=MC_BR_InitModPos_0.Done;
		MC_BR_InitModPos_0();

	(******************** INIT ENDLESS POSITION *********************)
		MC_BR_InitEndlessPosition_0.Execute:= InitModPos_Done;
		MC_BR_InitEndlessPosition_0.Axis:= gA[5].Ident;
		MC_BR_InitEndlessPosition_0.DataAddress:= ADR(gEndPosData[5]);
		IF (MC_BR_InitEndlessPosition_0.Done) THEN
			InitModPosition:=0;
			InitEndlessPosition:=0;
			HomeRestore:=1;
		END_IF
		MC_BR_InitEndlessPosition_0();

	(************************ HOME AXIS FIRST POWER UP **********************)
		IF (HomeRestore AND NOT gA5_FirstHomed) THEN
			MC_Home_0.Execute:=1;
		END_IF
		MC_Home_0.Axis:=gA[5].Ident;
		MC_Home_0.Position:=0;
		MC_Home_0.HomingMode:=mcHOME_DIRECT;
		IF (MC_Home_0.Done) THEN
			MC_Home_0.Execute:=0;
			gA5_FirstHomed:=1;
		END_IF
		MC_Home_0();

	(************************ HOME AXIS **********************)
		IF (gA5_FirstHomed) THEN
			MC_Home_1.Execute:=HomeRestore;
		END_IF
		MC_Home_1.Axis:=gA[5].Ident;
		MC_Home_1.Position:=0;
		MC_Home_1.HomingMode:=mcHOME_RESTORE_POS;
		IF (MC_Home_1.Done) THEN
			gA[5].Ind_Homed:=1;
			HomeRestore:=0;
		END_IF
		MC_Home_1();

	(******************** READ ACTUAL POSITION *********************)
		MC_ReadActualPosition_0.Enable:= gA[5].Ind_NetworkInit;
		MC_ReadActualPosition_0.Axis:= gA[5].Ident;
		MC_ReadActualPosition_0();
		IF(MC_ReadActualPosition_0.Valid = TRUE)THEN
			gA[5].PositionCount := MC_ReadActualPosition_0.Position;
			gA[5].PositionInch := gA[5].PositionCount/gA[5].UnitsPerInch;
			gA[5].PositionDeg := gA[5].PositionCount/gA[5].UnitsPerDeg;
		END_IF

	(******************** READ ACTUAL VELOCITY *********************)
		IF(MC_ReadActualVelocity_0.Error=TRUE) THEN
			MC_ReadActualVelocity_0.Enable:= 0;
		ELSE
			MC_ReadActualVelocity_0.Enable:= 1;
		END_IF
		MC_ReadActualVelocity_0.Axis:= gA[5].Ident;
		MC_ReadActualVelocity_0();
		IF(MC_ReadActualVelocity_0.Valid = TRUE)THEN
			//gA[5].ActualVelocity := MC_ReadActualVelocity_0.Velocity*60/gA[5].SP_MotorPPR;
      gA[5].ActualVelocity := MC_ReadActualVelocity_0.Velocity*60/gA[5].AxisPeriod ; // D.M. 03/08/2011 BrownPaper_14542  Need speed of the axis and not of the shaft of the motor
      IF ABS(gA[5].ActualVelocity>1) THEN // D.M. 03/08/2011 BrownPaper_14542 Add ABS because in case negative velocity Ind_InMotion = 0 instead of 1
				gA[5].Ind_InMotion:=1;
			ELSE
				gA[5].Ind_InMotion:=0;
			END_IF
		END_IF

	(******************** READ ACTUAL TORQUE *********************)
		IF(MC_ReadActualTorque_0.Error=TRUE) THEN
			MC_ReadActualTorque_0.Enable:= 0;
		ELSE
			MC_ReadActualTorque_0.Enable:= 1;
		END_IF
		MC_ReadActualTorque_0.Axis:= gA[5].Ident;
		MC_ReadActualTorque_0();
		IF(MC_ReadActualTorque_0.Valid = TRUE)THEN
			gA[5].ActualTorque := MC_ReadActualTorque_0.Torque;
		END_IF

	(************************ ENABLE AXIS **********************)
		MC_Power_0.Axis:=gA[5].Ident;
		IF (MC_Power_0.Error=0) THEN
			MC_Power_0.Enable:=gA[5].Cmd_Enable;
		ELSE;
			MC_Power_0.Enable:=0;
		END_IF;
		MC_Power_0();

	(************************ AXIS VELOCITY MOVE **********************)
		MC_MoveVelocity_0.Axis:=gA[5].Ident;
		MC_MoveVelocity_0.Velocity:=gA[5].SP_Velocity*gA[5].AxisPeriod/60;
		MC_MoveVelocity_0.Acceleration:=gA[5].SP_Accel;
		MC_MoveVelocity_0.Deceleration:=gA[5].SP_Decel;
		MC_MoveVelocity_0.Direction:=mcPOSITIVE_DIR;
		IF ((EDGEPOS(gA[5].Cmd_ContinuousMotion)) OR (EDGEPOS(gA[5].Cmd_ContinuousMotionUpdate))) THEN
			MC_MoveVelocity_0.Execute:=1;
		ELSE
			MC_MoveVelocity_0.Execute:=0;
		END_IF;
		MC_MoveVelocity_0();

  //************************ AXIS OVERRIDE **********************
    MC_SetOverride_0.Axis      := gA[5].Ident ;
    MC_SetOverride_0.Enable    := gA[5].Cmd_Override ;
    MC_SetOverride_0.VelFactor := gA[5].rSP_OverrideV ;
    MC_SetOverride_0.AccFactor := gA[5].rSP_OverrideA ;
    IF (MC_SetOverride_0.Enabled) OR
       (MC_SetOverride_0.Error)   THEN
      gA[5].Cmd_Override := 0 ;
    END_IF
    MC_SetOverride_0();

	(************************ AXIS STOP **********************)
		MC_Stop_0.Axis:=gA[5].Ident;
		IF (gA[5].Ind_ContinuousMotion AND (NOT gA[5].Cmd_ContinuousMotion) AND gAlarmsOK) THEN
			MC_Stop_0.Deceleration:=gA[5].SP_Decel;
			MC_Stop_0.Execute:=1;
		END_IF;
		IF (MC_Stop_0.Done OR MC_Stop_0.CommandAborted OR MC_Stop_0.Error) THEN
			MC_Stop_0.Execute:=0;
		END_IF;
		MC_Stop_0();

  (************************  ESTOP **********************)
    MC_Stop_1.Axis:=gA[5].Ident;
    IF EDGEPOS(g_bIndEStopStandstill) THEN
      MC_Stop_1.Deceleration:=gA[5].SP_EStopDecel;
      MC_Stop_1.Execute:=1;
    END_IF;
    IF (MC_Stop_1.Done OR MC_Stop_1.CommandAborted OR MC_Stop_1.Error) THEN
      MC_Stop_1.Execute:=0;
      gA[5].Cmd_EStopDisable := 1 ;
    END_IF;
    IF NOT(g_bIndEStopStandstill) THEN
      gA[5].Cmd_EStopDisable := 0 ;
    END_IF;
    MC_Stop_1();

		(************************ AXIS PHASE CONTROL (Inches) **********************)
		(*MC_BR_Phasing_0.Slave:=gA[5].Ident;
		IF (gA[5].Ind_SynchronizedMotion) THEN
			MC_BR_Phasing_0.Enable:=0;
		ELSE;
			MC_BR_Phasing_0.Enable:=0;
		END_IF;
		IF (gA[5].Cmd_PhaseOffset) THEN
			MC_BR_Phasing_0.InitData:=1;
			gA[5].Cmd_PhaseOffset:=0;
		ELSE
			MC_BR_Phasing_0.InitData:=0;
		END_IF
		MC_BR_Phasing_0.ApplicationMode:=mcMASTER_DISTANCE_BASED;
		MC_BR_Phasing_0.Shift:=gA[5].SP_PhaseOffset*gA[9].UnitsPerInch;
		MC_BR_Phasing_0.Velocity:=6*gA[5].AxisPeriod/60;
		MC_BR_Phasing_0.Acceleration:=gA[5].SP_Decel;
		MC_BR_Phasing_0.ApplicationDistance:=2*gA[9].AxisPeriod;
		MC_BR_Phasing_0.ShiftMode:=mcRELATIVE;
		MC_BR_Phasing_0();*)

	END_IF

END_PROGRAM
```

#### A5_Basic.var - Local variables
```iecst
(********************************************************************
 * COPYRIGHT -- Microsoft
 ********************************************************************
 * Program: A5_Basic
 * File: A5_Basic.var
 * Author: pkiel
 * Created: July 13, 2011
 ********************************************************************
 * Local variables of program A5_Basic
 ********************************************************************)
VAR
	AutoAck : BOOL;
	AxisErrorNcAccess : UINT;
	DriveStatus : MC_DRIVESTATUS_TYP;
	HomeRestore : BOOL;
	InitEndlessPosition : BOOL;
	InitModPos_Done : BOOL;
	InitModPosition : BOOL;
	MC_BR_InitEndlessPosition_0 : MC_BR_InitEndlessPosition;
	MC_BR_InitModPos_0 : MC_BR_InitModPos;
	(*MC_BR_Phasing_0 : MC_BR_Phasing;*)
	MC_BR_ReadDriveStatus_0 : MC_BR_ReadDriveStatus;
	MC_Home_0 : MC_Home;
	MC_Home_1 : MC_Home;
	MC_MoveVelocity_0 : MC_MoveVelocity;
	MC_Power_0 : MC_Power;
	MC_ReadActualPosition_0 : MC_ReadActualPosition;
	MC_ReadActualTorque_0 : MC_ReadActualTorque;
	MC_ReadActualVelocity_0 : MC_ReadActualVelocity;
	MC_ReadAxisError_0 : MC_ReadAxisError;
	MC_ReadStatus_0 : MC_ReadStatus;
	MC_Reset_0 : MC_Reset;
  MC_Stop_0 : MC_Stop;
  MC_Stop_1 : MC_Stop;
	ResetError : BOOL;
  MC_SetOverride_0 : MC_SetOverride;
END_VAR
```

### Program Logical/BagMachine_Section/EntryPull/Axis5/A5_Control (IEC) - Servo Control

#### A5_ControlCyclic.ld - Cyclic code
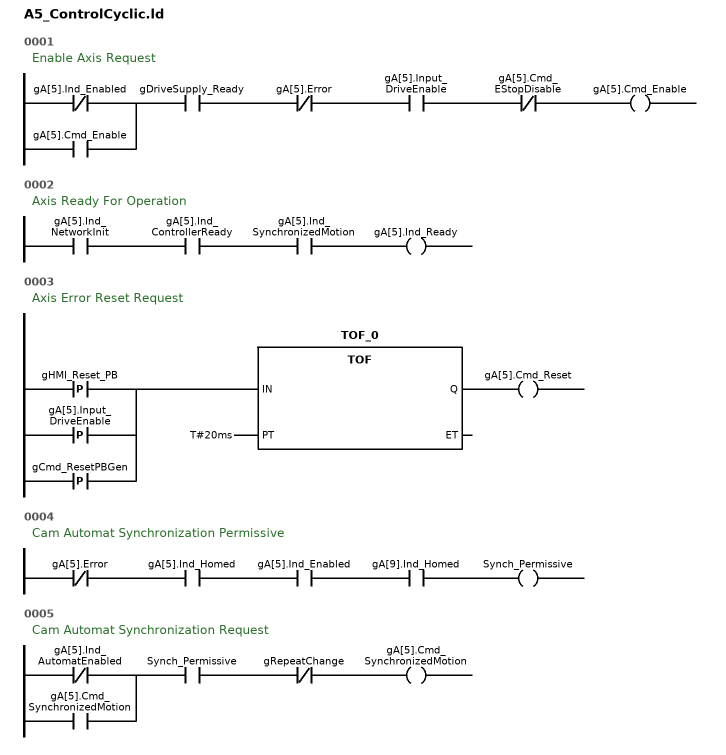
Ladder, written as Structured Text:
```iecst
(********************************************************************
 * COPYRIGHT -- Microsoft
 ********************************************************************
 * Program: A5_Control
 * File: A5_ControlCyclic.ld
 * Author: pkiel
 * Created: July 13, 2011
 ********************************************************************
 * Implementation of program A5_Control
 ********************************************************************)

PROGRAM _CYCLIC
VAR
    _e1 : R_TRIG;
    _e2 : R_TRIG;
    _e3 : R_TRIG;
END_VAR
(* Network 1: Enable Axis Request *)
gA[5].Cmd_Enable := (NOT gA[5].Ind_Enabled OR gA[5].Cmd_Enable) AND gDriveSupply_Ready AND NOT gA[5].Error AND gA[5].Input_DriveEnable AND NOT gA[5].Cmd_EStopDisable;

(* Network 2: Axis Ready For Operation *)
gA[5].Ind_Ready := gA[5].Ind_NetworkInit AND gA[5].Ind_ControllerReady AND gA[5].Ind_SynchronizedMotion;

(* Network 3: Axis Error Reset Request *)
_e1(CLK := gHMI_Reset_PB);
_e2(CLK := gA[5].Input_DriveEnable);
_e3(CLK := gCmd_ResetPBGen);
TOF_0(IN := _e1.Q OR _e2.Q OR _e3.Q, PT := T#20ms);
gA[5].Cmd_Reset := TOF_0.Q;

(* Network 4: Cam Automat Synchronization Permissive *)
Synch_Permissive := NOT gA[5].Error AND gA[5].Ind_Homed AND gA[5].Ind_Enabled AND gA[9].Ind_Homed;

(* Network 5: Cam Automat Synchronization Request *)
gA[5].Cmd_SynchronizedMotion := (NOT gA[5].Ind_AutomatEnabled OR gA[5].Cmd_SynchronizedMotion) AND Synch_Permissive AND NOT gRepeatChange;
END_PROGRAM
```

#### A5_Control.var - Local variables
```iecst
(********************************************************************
 * COPYRIGHT -- Microsoft
 ********************************************************************
 * Program: A5_Control
 * File: A5_Control.var
 * Author: pkiel
 * Created: July 13, 2011
 ********************************************************************
 * Local variables of program A5_Control
 ********************************************************************)
VAR
	Synch_Permissive : BOOL;
	TOF_0 : TOF;
END_VAR
```

### Program Logical/BagMachine_Section/EntryPull/Axis5/A5_Automat (IEC) - Cam Automat
